LIN {X 0,Y 392.107,Z 460.199,A -85,B 0,C 180,E1 -19978.685,E2 -19978.685} C_VEL
LIN {X 0,Y 391.923,Z 458.619,A -85,B 0,C 180,E1 -19981.316,E2 -19981.316} C_VEL
LIN {X 0,Y 395.453,Z 464.321,A -85,B 0,C 180,E1 -19989.606,E2 -19989.606} C_VEL
LIN {X 0,Y 398.852,Z 469.35,A -85,B 0,C 180,E1 -19992.892,E2 -19992.892} C_VEL
LIN {X 0,Y 400.055,Z 470.705,A -85,B 0,C 180,E1 -19993.809,E2 -19993.809} C_VEL
LIN {X 0,Y 404.204,Z 476.438,A -85,B 0,C 180,E1 -19996.602,E2 -19996.602} C_VEL
LIN {X 0,Y 408.109,Z 481.813,A -85,B 0,C 180,E1 -19998.795,E2 -19998.795} C_VEL
LIN {X 0,Y 412.144,Z 487.49,A -85,B 0,C 180,E1 -20000.782,E2 -20000.782} C_VEL
LIN {X 0,Y 417.683,Z 495.416,A -85,B 0,C 180,E1 -20003.182,E2 -20003.182} C_VEL
LIN {X 0,Y 425.779,Z 507.797,A -85,B 0,C 180,E1 -20006.237,E2 -20006.237} C_VEL
LIN {X 0,Y 433.973,Z 521.148,A -85,B 0,C 180,E1 -20008.937,E2 -20008.937} C_VEL
LIN {X 0,Y 436.683,Z 526.126,A -85,B 0,C 180,E1 -20009.777,E2 -20009.777} C_VEL
LIN {X 0,Y 420.829,Z 746.012,A -85,B 0,C 180,E1 -20013.375,E2 -20013.375} C_VEL
LIN {X 0,Y 417.528,Z 772.58,A -85,B 0,C 180,E1 -20013.976,E2 -20013.976} C_VEL
LIN {X 0,Y 413.994,Z 793.305,A -85,B 0,C 180,E1 -20014.607,E2 -20014.607} C_VEL
LIN {X 0,Y 408.88,Z 817.43,A -85,B 0,C 180,E1 -20015.544,E2 -20015.544} C_VEL
LIN {X 0,Y 403.422,Z 838.547,A -85,B 0,C 180,E1 -20016.579,E2 -20016.579} C_VEL
LIN {X 0,Y 396.748,Z 861.148,A -85,B 0,C 180,E1 -20017.924,E2 -20017.924} C_VEL
LIN {X 0,Y 389.639,Z 881.774,A -85,B 0,C 180,E1 -20019.428,E2 -20019.428} C_VEL
LIN {X 0,Y 382.034,Z 901.996,A -85,B 0,C 180,E1 -20021.184,E2 -20021.184} C_VEL
LIN {X 0,Y 373.957,Z 921.227,A -85,B 0,C 180,E1 -20023.196,E2 -20023.196} C_VEL
LIN {X 0,Y 366.455,Z 937.947,A -85,B 0,C 180,E1 -20025.254,E2 -20025.254} C_VEL
LIN {X 0,Y 357.859,Z 955.928,A -85,B 0,C 180,E1 -20027.888,E2 -20027.888} C_VEL
LIN {X 0,Y 350.795,Z 969.964,A -85,B 0,C 180,E1 -20030.322,E2 -20030.322} C_VEL
LIN {X 0,Y 343.188,Z 984.792,A -85,B 0,C 180,E1 -20033.325,E2 -20033.325} C_VEL
LIN {X 0,Y 336.074,Z 998.178,A -85,B 0,C 180,E1 -20036.605,E2 -20036.605} C_VEL
LIN {X 0,Y 329.965,Z 1009.92,A -85,B 0,C 180,E1 -20040,E2 -20040} C_VEL
LIN {X 0,Y 324.125,Z 1021.359,A -85,B 0,C 180,E1 -20044.02,E2 -20044.02} C_VEL
LIN {X 0,Y 319.921,Z 1030.19,A -85,B 0,C 180,E1 -20047.779,E2 -20047.779} C_VEL
LIN {X 0,Y 316.256,Z 1038.778,A -85,B 0,C 180,E1 -20052.331,E2 -20052.331} C_VEL
LIN {X 0,Y 314.196,Z 1044.51,A -85,B 0,C 180,E1 -20056.192,E2 -20056.192} C_VEL
LIN {X 0,Y 312.799,Z 1049.554,A -85,B 0,C 180,E1 -20060.617,E2 -20060.617} C_VEL
LIN {X 0,Y 312.21,Z 1052.658,A -85,B 0,C 180,E1 -20064.671,E2 -20064.671} C_VEL
LIN {X 0,Y 312.029,Z 1054.407,A -85,B 0,C 180,E1 -20068.347,E2 -20068.347} C_VEL
LIN {X 0,Y 311.984,Z 1055.15,A -85,B 0,C 180,E1 -20072.204,E2 -20072.204} C_VEL
LIN {X 0,Y 312.068,Z 1054.525,A -85,B 0,C 180,E1 -20076.439,E2 -20076.439} C_VEL
LIN {X 0,Y 312.31,Z 1052.851,A -85,B 0,C 180,E1 -20080.142,E2 -20080.142} C_VEL
LIN {X 0,Y 312.996,Z 1049.964,A -85,B 0,C 180,E1 -20084.051,E2 -20084.051} C_VEL
LIN {X 0,Y 314.708,Z 1044.785,A -85,B 0,C 180,E1 -20088.771,E2 -20088.771} C_VEL
LIN {X 0,Y 317.043,Z 1039.138,A -85,B 0,C 180,E1 -20092.629,E2 -20092.629} C_VEL
LIN {X 0,Y 320.972,Z 1030.962,A -85,B 0,C 180,E1 -20097.053,E2 -20097.053} C_VEL
LIN {X 0,Y 325.565,Z 1022.129,A -85,B 0,C 180,E1 -20100.857,E2 -20100.857} C_VEL
LIN {X 0,Y 331.629,Z 1011.288,A -85,B 0,C 180,E1 -20104.74,E2 -20104.74} C_VEL
LIN {X 0,Y 338.541,Z 998.922,A -85,B 0,C 180,E1 -20108.334,E2 -20108.334} C_VEL
LIN {X 0,Y 346.21,Z 985.46,A -85,B 0,C 180,E1 -20111.626,E2 -20111.626} C_VEL
LIN {X 0,Y 354.624,Z 970.07,A -85,B 0,C 180,E1 -20114.721,E2 -20114.721} C_VEL
LIN {X 0,Y 363.408,Z 953.602,A -85,B 0,C 180,E1 -20117.509,E2 -20117.509} C_VEL
LIN {X 0,Y 372.16,Z 935.987,A -85,B 0,C 180,E1 -20119.971,E2 -20119.971} C_VEL
LIN {X 0,Y 380.693,Z 917.814,A -85,B 0,C 180,E1 -20122.117,E2 -20122.117} C_VEL
LIN {X 0,Y 389.097,Z 898.152,A -85,B 0,C 180,E1 -20124.045,E2 -20124.045} C_VEL
LIN {X 0,Y 396.341,Z 879.576,A -85,B 0,C 180,E1 -20125.584,E2 -20125.584} C_VEL
LIN {X 0,Y 404.502,Z 856.112,A -85,B 0,C 180,E1 -20127.187,E2 -20127.187} C_VEL
LIN {X 0,Y 408.136,Z 844.614,A -85,B 0,C 180,E1 -20127.862,E2 -20127.862} C_VEL
LIN {X 0,Y 409.545,Z 837.786,A -85,B 0,C 180,E1 -20128.344,E2 -20128.344} C_VEL
LIN {X 0,Y 411.055,Z 821.016,A -85,B 0,C 180,E1 -20129.882,E2 -20129.882} C_VEL
LIN {X 0,Y 412.236,Z 813.969,A -85,B 0,C 180,E1 -20130.298,E2 -20130.298} C_VEL
LIN {X 0,Y 417.189,Z 791.229,A -85,B 0,C 180,E1 -20131.12,E2 -20131.12} C_VEL
LIN {X 0,Y 421.292,Z 767.977,A -85,B 0,C 180,E1 -20131.778,E2 -20131.778} C_VEL
LIN {X 0,Y 424.228,Z 743.452,A -85,B 0,C 180,E1 -20132.284,E2 -20132.284} C_VEL
LIN {X 0,Y 440.243,Z 535.419,A -85,B 0,C 180,E1 -20135.639,E2 -20135.639} C_VEL
LIN {X 0,Y 432.705,Z 522.887,A -85,B 0,C 180,E1 -20138.372,E2 -20138.372} C_VEL
LIN {X 0,Y 425.772,Z 512.089,A -85,B 0,C 180,E1 -20141.268,E2 -20141.268} C_VEL
LIN {X 0,Y 420.737,Z 504.576,A -85,B 0,C 180,E1 -20143.714,E2 -20143.714} C_VEL
LIN {X 0,Y 417.623,Z 500.075,A -85,B 0,C 180,E1 -20145.44,E2 -20145.44} C_VEL
LIN {X 0,Y 414.64,Z 495.722,A -85,B 0,C 180,E1 -20147.324,E2 -20147.324} C_VEL
LIN {X 0,Y 411.54,Z 491.193,A -85,B 0,C 180,E1 -20149.642,E2 -20149.642} C_VEL
LIN {X 0,Y 408.5,Z 486.912,A -85,B 0,C 180,E1 -20152.546,E2 -20152.546} C_VEL
LIN {X 0,Y 407.925,Z 485.949,A -85,B 0,C 180,E1 -20153.243,E2 -20153.243} C_VEL
LIN {X 0,Y 404.96,Z 480.934,A -85,B 0,C 180,E1 -20160.707,E2 -20160.707} C_VEL
LIN {X 0,Y 405.174,Z 482.493,A -85,B 0,C 180,E1 -20163.395,E2 -20163.395} C_VEL
LIN {X 0,Y 408.31,Z 486.414,A -85,B 0,C 180,E1 -20168.875,E2 -20168.875} C_VEL
LIN {X 0,Y 410.739,Z 490.415,A -85,B 0,C 180,E1 -20171.372,E2 -20171.372} C_VEL
LIN {X 0,Y 412.175,Z 492.139,A -85,B 0,C 180,E1 -20172.54,E2 -20172.54} C_VEL
LIN {X 0,Y 416.043,Z 497.712,A -85,B 0,C 180,E1 -20175.258,E2 -20175.258} C_VEL
LIN {X 0,Y 419.58,Z 502.842,A -85,B 0,C 180,E1 -20177.331,E2 -20177.331} C_VEL
LIN {X 0,Y 423.084,Z 508.142,A -85,B 0,C 180,E1 -20179.142,E2 -20179.142} C_VEL
LIN {X 0,Y 430.274,Z 520.703,A -85,B 0,C 180,E1 -20182.403,E2 -20182.403} C_VEL
LIN {X 0,Y 438.135,Z 535.607,A -85,B 0,C 180,E1 -20185.443,E2 -20185.443} C_VEL
LIN {X 0,Y 440.062,Z 539.907,A -85,B 0,C 180,E1 -20186.145,E2 -20186.145} C_VEL
LIN {X 0,Y 423.319,Z 757.439,A -85,B 0,C 180,E1 -20189.661,E2 -20189.661} C_VEL
LIN {X 0,Y 419.717,Z 784.19,A -85,B 0,C 180,E1 -20190.228,E2 -20190.228} C_VEL
LIN {X 0,Y 415.608,Z 805.997,A -85,B 0,C 180,E1 -20190.833,E2 -20190.833} C_VEL
LIN {X 0,Y 409.689,Z 831.066,A -85,B 0,C 180,E1 -20191.743,E2 -20191.743} C_VEL
LIN {X 0,Y 403.918,Z 851.482,A -85,B 0,C 180,E1 -20192.684,E2 -20192.684} C_VEL
LIN {X 0,Y 396.612,Z 874.086,A -85,B 0,C 180,E1 -20193.959,E2 -20193.959} C_VEL
LIN {X 0,Y 389.187,Z 894.048,A -85,B 0,C 180,E1 -20195.342,E2 -20195.342} C_VEL
LIN {X 0,Y 381.105,Z 913.869,A -85,B 0,C 180,E1 -20196.974,E2 -20196.974} C_VEL
LIN {X 0,Y 372.228,Z 933.564,A -85,B 0,C 180,E1 -20198.946,E2 -20198.946} C_VEL
LIN {X 0,Y 364.051,Z 950.448,A -85,B 0,C 180,E1 -20200.948,E2 -20200.948} C_VEL
LIN {X 0,Y 354.07,Z 969.767,A -85,B 0,C 180,E1 -20203.702,E2 -20203.702} C_VEL
LIN {X 0,Y 345.849,Z 984.889,A -85,B 0,C 180,E1 -20206.292,E2 -20206.292} C_VEL
LIN {X 0,Y 336.675,Z 1001.243,A -85,B 0,C 180,E1 -20209.651,E2 -20209.651} C_VEL
LIN {X 0,Y 329.367,Z 1014.076,A -85,B 0,C 180,E1 -20212.834,E2 -20212.834} C_VEL
LIN {X 0,Y 322.102,Z 1027.018,A -85,B 0,C 180,E1 -20216.67,E2 -20216.67} C_VEL
LIN {X 0,Y 316.389,Z 1037.489,A -85,B 0,C 180,E1 -20220.461,E2 -20220.461} C_VEL
LIN {X 0,Y 311.489,Z 1047.292,A -85,B 0,C 180,E1 -20224.727,E2 -20224.727} C_VEL
LIN {X 0,Y 307.959,Z 1055.162,A -85,B 0,C 180,E1 -20229.075,E2 -20229.075} C_VEL
LIN {X 0,Y 305.682,Z 1061.542,A -85,B 0,C 180,E1 -20233.466,E2 -20233.466} C_VEL
LIN {X 0,Y 304.419,Z 1066.404,A -85,B 0,C 180,E1 -20238.058,E2 -20238.058} C_VEL
LIN {X 0,Y 304.013,Z 1069.246,A -85,B 0,C 180,E1 -20241.885,E2 -20241.885} C_VEL
LIN {X 0,Y 303.96,Z 1071.045,A -85,B 0,C 180,E1 -20245.85,E2 -20245.85} C_VEL
LIN {X 0,Y 304.002,Z 1071.567,A -85,B 0,C 180,E1 -20250,E2 -20250} C_VEL
LIN {X 0,Y 303.97,Z 1070.824,A -85,B 0,C 180,E1 -20253.772,E2 -20253.772} C_VEL
LIN {X 0,Y 304.002,Z 1069.099,A -85,B 0,C 180,E1 -20257.37,E2 -20257.37} C_VEL
LIN {X 0,Y 304.317,Z 1066.031,A -85,B 0,C 180,E1 -20261.37,E2 -20261.37} C_VEL
LIN {X 0,Y 305.49,Z 1060.637,A -85,B 0,C 180,E1 -20266.153,E2 -20266.153} C_VEL
LIN {X 0,Y 307.385,Z 1054.653,A -85,B 0,C 180,E1 -20270.17,E2 -20270.17} C_VEL
LIN {X 0,Y 310.78,Z 1046.13,A -85,B 0,C 180,E1 -20274.724,E2 -20274.724} C_VEL
LIN {X 0,Y 314.948,Z 1036.991,A -85,B 0,C 180,E1 -20278.646,E2 -20278.646} C_VEL
LIN {X 0,Y 320.569,Z 1025.802,A -85,B 0,C 180,E1 -20282.657,E2 -20282.657} C_VEL
LIN {X 0,Y 327.144,Z 1013.096,A -85,B 0,C 180,E1 -20286.366,E2 -20286.366} C_VEL
LIN {X 0,Y 334.671,Z 998.993,A -85,B 0,C 180,E1 -20289.84,E2 -20289.84} C_VEL
LIN {X 0,Y 342.892,Z 983.203,A -85,B 0,C 180,E1 -20293.028,E2 -20293.028} C_VEL
LIN {X 0,Y 351.564,Z 966.327,A -85,B 0,C 180,E1 -20295.901,E2 -20295.901} C_VEL
LIN {X 0,Y 359.956,Z 948.899,A -85,B 0,C 180,E1 -20298.351,E2 -20298.351} C_VEL
LIN {X 0,Y 367.87,Z 931.67,A -85,B 0,C 180,E1 -20300.41,E2 -20300.41} C_VEL
LIN {X 0,Y 376.774,Z 910.555,A -85,B 0,C 180,E1 -20302.513,E2 -20302.513} C_VEL
LIN {X 0,Y 383.859,Z 892.297,A -85,B 0,C 180,E1 -20304.028,E2 -20304.028} C_VEL
LIN {X 0,Y 391.912,Z 869.15,A -85,B 0,C 180,E1 -20305.624,E2 -20305.624} C_VEL
LIN {X 0,Y 397.756,Z 850.018,A -85,B 0,C 180,E1 -20306.704,E2 -20306.704} C_VEL
LIN {X 0,Y 403.893,Z 827.253,A -85,B 0,C 180,E1 -20307.764,E2 -20307.764} C_VEL
LIN {X 0,Y 409.005,Z 803.859,A -85,B 0,C 180,E1 -20308.606,E2 -20308.606} C_VEL
LIN {X 0,Y 413.132,Z 780.688,A -85,B 0,C 180,E1 -20309.254,E2 -20309.254} C_VEL
LIN {X 0,Y 416.173,Z 755.582,A -85,B 0,C 180,E1 -20309.781,E2 -20309.781} C_VEL
LIN {X 0,Y 432.44,Z 534.422,A -85,B 0,C 180,E1 -20313.402,E2 -20313.402} C_VEL
LIN {X 0,Y 425.765,Z 521.335,A -85,B 0,C 180,E1 -20315.66,E2 -20315.66} C_VEL
LIN {X 0,Y 419.365,Z 509.666,A -85,B 0,C 180,E1 -20318.054,E2 -20318.054} C_VEL
LIN {X 0,Y 413.828,Z 500.099,A -85,B 0,C 180,E1 -20320.376,E2 -20320.376} C_VEL
LIN {X 0,Y 408.544,Z 492.288,A -85,B 0,C 180,E1 -20322.847,E2 -20322.847} C_VEL
LIN {X 0,Y 404.593,Z 486.761,A -85,B 0,C 180,E1 -20324.96,E2 -20324.96} C_VEL
LIN {X 0,Y 401.658,Z 482.574,A -85,B 0,C 180,E1 -20326.76,E2 -20326.76} C_VEL
LIN {X 0,Y 397.969,Z 477.456,A -85,B 0,C 180,E1 -20329.431,E2 -20329.431} C_VEL
LIN {X 0,Y 395.072,Z 473.702,A -85,B 0,C 180,E1 -20332.072,E2 -20332.072} C_VEL
LIN {X 0,Y 394.278,Z 472.195,A -85,B 0,C 180,E1 -20333.008,E2 -20333.008} C_VEL
LIN {X 0,Y 390.943,Z 466.591,A -85,B 0,C 180,E1 -20341.172,E2 -20341.172} C_VEL
LIN {X 0,Y 391.332,Z 468.804,A -85,B 0,C 180,E1 -20344.543,E2 -20344.543} C_VEL
LIN {X 0,Y 394.595,Z 472.62,A -85,B 0,C 180,E1 -20349.775,E2 -20349.775} C_VEL
LIN {X 0,Y 397.351,Z 476.896,A -85,B 0,C 180,E1 -20352.498,E2 -20352.498} C_VEL
LIN {X 0,Y 398.703,Z 478.42,A -85,B 0,C 180,E1 -20353.561,E2 -20353.561} C_VEL
LIN {X 0,Y 402.767,Z 484.173,A -85,B 0,C 180,E1 -20356.366,E2 -20356.366} C_VEL
LIN {X 0,Y 406.481,Z 489.377,A -85,B 0,C 180,E1 -20358.501,E2 -20358.501} C_VEL
LIN {X 0,Y 410.443,Z 495.07,A -85,B 0,C 180,E1 -20360.499,E2 -20360.499} C_VEL
LIN {X 0,Y 415.829,Z 502.974,A -85,B 0,C 180,E1 -20362.889,E2 -20362.889} C_VEL
LIN {X 0,Y 423.519,Z 514.987,A -85,B 0,C 180,E1 -20365.86,E2 -20365.86} C_VEL
LIN {X 0,Y 431.288,Z 527.889,A -85,B 0,C 180,E1 -20368.49,E2 -20368.49} C_VEL
LIN {X 0,Y 432.587,Z 530.46,A -85,B 0,C 180,E1 -20368.913,E2 -20368.913} C_VEL
LIN {X 0,Y 416.611,Z 746.198,A -85,B 0,C 180,E1 -20372.444,E2 -20372.444} C_VEL
LIN {X 0,Y 413.237,Z 772.776,A -85,B 0,C 180,E1 -20373.044,E2 -20373.044} C_VEL
LIN {X 0,Y 409.644,Z 793.399,A -85,B 0,C 180,E1 -20373.668,E2 -20373.668} C_VEL
LIN {X 0,Y 404.466,Z 817.349,A -85,B 0,C 180,E1 -20374.592,E2 -20374.592} C_VEL
LIN {X 0,Y 399.02,Z 837.987,A -85,B 0,C 180,E1 -20375.595,E2 -20375.595} C_VEL
LIN {X 0,Y 392.484,Z 859.751,A -85,B 0,C 180,E1 -20376.875,E2 -20376.875} C_VEL
LIN {X 0,Y 385.178,Z 880.634,A -85,B 0,C 180,E1 -20378.375,E2 -20378.375} C_VEL
LIN {X 0,Y 378.164,Z 898.884,A -85,B 0,C 180,E1 -20379.935,E2 -20379.935} C_VEL
LIN {X 0,Y 369.204,Z 920.008,A -85,B 0,C 180,E1 -20382.093,E2 -20382.093} C_VEL
LIN {X 0,Y 361.513,Z 936.692,A -85,B 0,C 180,E1 -20384.132,E2 -20384.132} C_VEL
LIN {X 0,Y 352.516,Z 955.067,A -85,B 0,C 180,E1 -20386.8,E2 -20386.8} C_VEL
LIN {X 0,Y 344.576,Z 970.313,A -85,B 0,C 180,E1 -20389.458,E2 -20389.458} C_VEL
LIN {X 0,Y 336.694,Z 985.124,A -85,B 0,C 180,E1 -20392.498,E2 -20392.498} C_VEL
LIN {X 0,Y 328.953,Z 999.119,A -85,B 0,C 180,E1 -20395.993,E2 -20395.993} C_VEL
LIN {X 0,Y 322.348,Z 1011.352,A -85,B 0,C 180,E1 -20399.628,E2 -20399.628} C_VEL
LIN {X 0,Y 316.58,Z 1022.099,A -85,B 0,C 180,E1 -20403.555,E2 -20403.555} C_VEL
LIN {X 0,Y 312.039,Z 1031.265,A -85,B 0,C 180,E1 -20407.585,E2 -20407.585} C_VEL
LIN {X 0,Y 308.405,Z 1039.339,A -85,B 0,C 180,E1 -20412.061,E2 -20412.061} C_VEL
LIN {X 0,Y 306.264,Z 1045.015,A -85,B 0,C 180,E1 -20416.019,E2 -20416.019} C_VEL
LIN {X 0,Y 304.773,Z 1050.105,A -85,B 0,C 180,E1 -20420.749,E2 -20420.749} C_VEL
LIN {X 0,Y 304.21,Z 1053,A -85,B 0,C 180,E1 -20424.72,E2 -20424.72} C_VEL
LIN {X 0,Y 304.03,Z 1054.698,A -85,B 0,C 180,E1 -20428.492,E2 -20428.492} C_VEL
LIN {X 0,Y 303.99,Z 1055.394,A -85,B 0,C 180,E1 -20432.639,E2 -20432.639} C_VEL
LIN {X 0,Y 304.084,Z 1054.663,A -85,B 0,C 180,E1 -20436.798,E2 -20436.798} C_VEL
LIN {X 0,Y 304.342,Z 1053.049,A -85,B 0,C 180,E1 -20440.41,E2 -20440.41} C_VEL
LIN {X 0,Y 305.096,Z 1050.156,A -85,B 0,C 180,E1 -20444.423,E2 -20444.423} C_VEL
LIN {X 0,Y 306.918,Z 1045.034,A -85,B 0,C 180,E1 -20449.211,E2 -20449.211} C_VEL
LIN {X 0,Y 309.449,Z 1039.309,A -85,B 0,C 180,E1 -20453.216,E2 -20453.216} C_VEL
LIN {X 0,Y 313.625,Z 1031.117,A -85,B 0,C 180,E1 -20457.741,E2 -20457.741} C_VEL
LIN {X 0,Y 318.474,Z 1022.276,A -85,B 0,C 180,E1 -20461.622,E2 -20461.622} C_VEL
LIN {X 0,Y 324.84,Z 1011.42,A -85,B 0,C 180,E1 -20465.574,E2 -20465.574} C_VEL
LIN {X 0,Y 332.074,Z 999.042,A -85,B 0,C 180,E1 -20469.222,E2 -20469.222} C_VEL
LIN {X 0,Y 340.062,Z 985.569,A -85,B 0,C 180,E1 -20472.553,E2 -20472.553} C_VEL
LIN {X 0,Y 348.532,Z 970.629,A -85,B 0,C 180,E1 -20475.59,E2 -20475.59} C_VEL
LIN {X 0,Y 356.861,Z 955.523,A -85,B 0,C 180,E1 -20478.185,E2 -20478.185} C_VEL
LIN {X 0,Y 366.378,Z 937.141,A -85,B 0,C 180,E1 -20480.811,E2 -20480.811} C_VEL
LIN {X 0,Y 374.547,Z 920.273,A -85,B 0,C 180,E1 -20482.833,E2 -20482.833} C_VEL
LIN {X 0,Y 384.052,Z 898.875,A -85,B 0,C 180,E1 -20484.966,E2 -20484.966} C_VEL
LIN {X 0,Y 391.16,Z 881.166,A -85,B 0,C 180,E1 -20486.442,E2 -20486.442} C_VEL
LIN {X 0,Y 399.138,Z 859.19,A -85,B 0,C 180,E1 -20487.973,E2 -20487.973} C_VEL
LIN {X 0,Y 405.748,Z 837.99,A -85,B 0,C 180,E1 -20489.183,E2 -20489.183} C_VEL
LIN {X 0,Y 411.995,Z 815.05,A -85,B 0,C 180,E1 -20490.255,E2 -20490.255} C_VEL
LIN {X 0,Y 412.236,Z 813.969,A -85,B 0,C 180,E1 -20490.298,E2 -20490.298} C_VEL
LIN {X 0,Y 413.356,Z 806.832,A -85,B 0,C 180,E1 -20490.698,E2 -20490.698} C_VEL
LIN {X 0,Y 414.24,Z 789.235,A -85,B 0,C 180,E1 -20492.044,E2 -20492.044} C_VEL
LIN {X 0,Y 415.089,Z 781.926,A -85,B 0,C 180,E1 -20492.378,E2 -20492.378} C_VEL
LIN {X 0,Y 418.675,Z 758.825,A -85,B 0,C 180,E1 -20492.947,E2 -20492.947} C_VEL
LIN {X 0,Y 421.397,Z 733.209,A -85,B 0,C 180,E1 -20493.422,E2 -20493.422} C_VEL
LIN {X 0,Y 436.472,Z 540.091,A -85,B 0,C 180,E1 -20496.527,E2 -20496.527} C_VEL
LIN {X 0,Y 430.16,Z 529.414,A -85,B 0,C 180,E1 -20498.917,E2 -20498.917} C_VEL
LIN {X 0,Y 423.64,Z 519,A -85,B 0,C 180,E1 -20501.74,E2 -20501.74} C_VEL
LIN {X 0,Y 418.868,Z 511.764,A -85,B 0,C 180,E1 -20504.138,E2 -20504.138} C_VEL
LIN {X 0,Y 415.843,Z 507.313,A -85,B 0,C 180,E1 -20505.874,E2 -20505.874} C_VEL
LIN {X 0,Y 413.255,Z 503.408,A -85,B 0,C 180,E1 -20507.564,E2 -20507.564} C_VEL
LIN {X 0,Y 410.054,Z 498.749,A -85,B 0,C 180,E1 -20510.03,E2 -20510.03} C_VEL
LIN {X 0,Y 407.172,Z 494.337,A -85,B 0,C 180,E1 -20512.947,E2 -20512.947} C_VEL
LIN {X 0,Y 403.983,Z 488.887,A -85,B 0,C 180,E1 -20520.709,E2 -20520.709} C_VEL
LIN {X 0,Y 404.263,Z 490.703,A -85,B 0,C 180,E1 -20523.687,E2 -20523.687} C_VEL
LIN {X 0,Y 407.205,Z 494.378,A -85,B 0,C 180,E1 -20528.757,E2 -20528.757} C_VEL
LIN {X 0,Y 409.769,Z 498.475,A -85,B 0,C 180,E1 -20531.4,E2 -20531.4} C_VEL
LIN {X 0,Y 410.93,Z 499.999,A -85,B 0,C 180,E1 -20532.364,E2 -20532.364} C_VEL
LIN {X 0,Y 414.531,Z 505.26,A -85,B 0,C 180,E1 -20534.957,E2 -20534.957} C_VEL
LIN {X 0,Y 417.988,Z 510.399,A -85,B 0,C 180,E1 -20537.04,E2 -20537.04} C_VEL
LIN {X 0,Y 421.29,Z 515.524,A -85,B 0,C 180,E1 -20538.795,E2 -20538.795} C_VEL
LIN {X 0,Y 428.233,Z 527.953,A -85,B 0,C 180,E1 -20542.034,E2 -20542.034} C_VEL
LIN {X 0,Y 435.709,Z 542.535,A -85,B 0,C 180,E1 -20545.013,E2 -20545.013} C_VEL
LIN {X 0,Y 436.342,Z 544.175,A -85,B 0,C 180,E1 -20545.261,E2 -20545.261} C_VEL
LIN {X 0,Y 419.514,Z 757.283,A -85,B 0,C 180,E1 -20548.7,E2 -20548.7} C_VEL
LIN {X 0,Y 415.84,Z 784.009,A -85,B 0,C 180,E1 -20549.263,E2 -20549.263} C_VEL
LIN {X 0,Y 411.668,Z 805.744,A -85,B 0,C 180,E1 -20549.862,E2 -20549.862} C_VEL
LIN {X 0,Y 405.695,Z 830.577,A -85,B 0,C 180,E1 -20550.753,E2 -20550.753} C_VEL
LIN {X 0,Y 399.826,Z 850.919,A -85,B 0,C 180,E1 -20551.68,E2 -20551.68} C_VEL
LIN {X 0,Y 392.489,Z 873.21,A -85,B 0,C 180,E1 -20552.921,E2 -20552.921} C_VEL
LIN {X 0,Y 384.643,Z 893.826,A -85,B 0,C 180,E1 -20554.34,E2 -20554.34} C_VEL
LIN {X 0,Y 376.465,Z 913.378,A -85,B 0,C 180,E1 -20555.943,E2 -20555.943} C_VEL
LIN {X 0,Y 367.131,Z 933.544,A -85,B 0,C 180,E1 -20557.958,E2 -20557.958} C_VEL
LIN {X 0,Y 358.732,Z 950.377,A -85,B 0,C 180,E1 -20559.959,E2 -20559.959} C_VEL
LIN {X 0,Y 348.439,Z 969.671,A -85,B 0,C 180,E1 -20562.725,E2 -20562.725} C_VEL
LIN {X 0,Y 340.417,Z 983.933,A -85,B 0,C 180,E1 -20565.175,E2 -20565.175} C_VEL
LIN {X 0,Y 331.284,Z 999.705,A -85,B 0,C 180,E1 -20568.394,E2 -20568.394} C_VEL
LIN {X 0,Y 323.557,Z 1012.659,A -85,B 0,C 180,E1 -20571.6,E2 -20571.6} C_VEL
LIN {X 0,Y 316.145,Z 1025.308,A -85,B 0,C 180,E1 -20575.318,E2 -20575.318} C_VEL
LIN {X 0,Y 309.724,Z 1036.399,A -85,B 0,C 180,E1 -20579.331,E2 -20579.331} C_VEL
LIN {X 0,Y 304.832,Z 1045.506,A -85,B 0,C 180,E1 -20583.296,E2 -20583.296} C_VEL
LIN {X 0,Y 300.554,Z 1054.364,A -85,B 0,C 180,E1 -20588.124,E2 -20588.124} C_VEL
LIN {X 0,Y 298.169,Z 1060.337,A -85,B 0,C 180,E1 -20592.247,E2 -20592.247} C_VEL
LIN {X 0,Y 296.588,Z 1065.714,A -85,B 0,C 180,E1 -20597.144,E2 -20597.144} C_VEL
LIN {X 0,Y 296.057,Z 1068.802,A -85,B 0,C 180,E1 -20601.258,E2 -20601.258} C_VEL
LIN {X 0,Y 295.965,Z 1070.558,A -85,B 0,C 180,E1 -20604.961,E2 -20604.961} C_VEL
LIN {X 0,Y 295.988,Z 1071.34,A -85,B 0,C 180,E1 -20608.839,E2 -20608.839} C_VEL
LIN {X 0,Y 295.982,Z 1070.949,A -85,B 0,C 180,E1 -20612.905,E2 -20612.905} C_VEL
LIN {X 0,Y 295.985,Z 1069.219,A -85,B 0,C 180,E1 -20616.985,E2 -20616.985} C_VEL
LIN {X 0,Y 296.236,Z 1066.514,A -85,B 0,C 180,E1 -20620.82,E2 -20620.82} C_VEL
LIN {X 0,Y 297.163,Z 1062.133,A -85,B 0,C 180,E1 -20625.216,E2 -20625.216} C_VEL
LIN {X 0,Y 299.206,Z 1055.636,A -85,B 0,C 180,E1 -20629.93,E2 -20629.93} C_VEL
LIN {X 0,Y 302.078,Z 1048.532,A -85,B 0,C 180,E1 -20634.025,E2 -20634.025} C_VEL
LIN {X 0,Y 306.759,Z 1038.581,A -85,B 0,C 180,E1 -20638.63,E2 -20638.63} C_VEL
LIN {X 0,Y 311.855,Z 1028.689,A -85,B 0,C 180,E1 -20642.374,E2 -20642.374} C_VEL
LIN {X 0,Y 319.086,Z 1015.375,A -85,B 0,C 180,E1 -20646.54,E2 -20646.54} C_VEL
LIN {X 0,Y 326.141,Z 1002.551,A -85,B 0,C 180,E1 -20649.848,E2 -20649.848} C_VEL
LIN {X 0,Y 334.628,Z 987.115,A -85,B 0,C 180,E1 -20653.19,E2 -20653.19} C_VEL
LIN {X 0,Y 342.594,Z 972.097,A -85,B 0,C 180,E1 -20655.887,E2 -20655.887} C_VEL
LIN {X 0,Y 351.575,Z 954.674,A -85,B 0,C 180,E1 -20658.539,E2 -20658.539} C_VEL
LIN {X 0,Y 360.377,Z 936.242,A -85,B 0,C 180,E1 -20660.85,E2 -20660.85} C_VEL
LIN {X 0,Y 368.441,Z 918.26,A -85,B 0,C 180,E1 -20662.758,E2 -20662.758} C_VEL
LIN {X 0,Y 377.103,Z 897.095,A -85,B 0,C 180,E1 -20664.621,E2 -20664.621} C_VEL
LIN {X 0,Y 384.111,Z 878.167,A -85,B 0,C 180,E1 -20666.006,E2 -20666.006} C_VEL
LIN {X 0,Y 391.773,Z 854.86,A -85,B 0,C 180,E1 -20667.417,E2 -20667.417} C_VEL
LIN {X 0,Y 397.76,Z 833.621,A -85,B 0,C 180,E1 -20668.449,E2 -20668.449} C_VEL
LIN {X 0,Y 403.532,Z 809.714,A -85,B 0,C 180,E1 -20669.379,E2 -20669.379} C_VEL
LIN {X 0,Y 407.972,Z 786.31,A -85,B 0,C 180,E1 -20670.064,E2 -20670.064} C_VEL
LIN {X 0,Y 411.49,Z 761.683,A -85,B 0,C 180,E1 -20670.621,E2 -20670.621} C_VEL
LIN {X 0,Y 415.66,Z 708.814,A -85,B 0,C 180,E1 -20671.518,E2 -20671.518} C_VEL
LIN {X 0,Y 428.389,Z 538.48,A -85,B 0,C 180,E1 -20674.303,E2 -20674.303} C_VEL
LIN {X 0,Y 422.76,Z 527.263,A -85,B 0,C 180,E1 -20676.292,E2 -20676.292} C_VEL
LIN {X 0,Y 416.946,Z 516.392,A -85,B 0,C 180,E1 -20678.548,E2 -20678.548} C_VEL
LIN {X 0,Y 411.771,Z 507.237,A -85,B 0,C 180,E1 -20680.79,E2 -20680.79} C_VEL
LIN {X 0,Y 406.611,Z 499.485,A -85,B 0,C 180,E1 -20683.279,E2 -20683.279} C_VEL
LIN {X 0,Y 402.77,Z 493.992,A -85,B 0,C 180,E1 -20685.405,E2 -20685.405} C_VEL
LIN {X 0,Y 400.136,Z 490.146,A -85,B 0,C 180,E1 -20687.076,E2 -20687.076} C_VEL
LIN {X 0,Y 396.634,Z 485.178,A -85,B 0,C 180,E1 -20689.689,E2 -20689.689} C_VEL
LIN {X 0,Y 393.764,Z 481.254,A -85,B 0,C 180,E1 -20692.412,E2 -20692.412} C_VEL
LIN {X 0,Y 393.175,Z 480.083,A -85,B 0,C 180,E1 -20693.135,E2 -20693.135} C_VEL
LIN {X 0,Y 389.968,Z 474.534,A -85,B 0,C 180,E1 -20701.175,E2 -20701.175} C_VEL
LIN {X 0,Y 390.545,Z 477.299,A -85,B 0,C 180,E1 -20705.141,E2 -20705.141} C_VEL
LIN {X 0,Y 393.421,Z 480.441,A -85,B 0,C 180,E1 -20709.575,E2 -20709.575} C_VEL
LIN {X 0,Y 396.332,Z 484.908,A -85,B 0,C 180,E1 -20712.487,E2 -20712.487} C_VEL
LIN {X 0,Y 397.53,Z 486.454,A -85,B 0,C 180,E1 -20713.454,E2 -20713.454} C_VEL
LIN {X 0,Y 401.23,Z 491.726,A -85,B 0,C 180,E1 -20716.059,E2 -20716.059} C_VEL
LIN {X 0,Y 404.987,Z 497.134,A -85,B 0,C 180,E1 -20718.274,E2 -20718.274} C_VEL
LIN {X 0,Y 408.822,Z 502.749,A -85,B 0,C 180,E1 -20720.248,E2 -20720.248} C_VEL
LIN {X 0,Y 414.357,Z 511.11,A -85,B 0,C 180,E1 -20722.75,E2 -20722.75} C_VEL
LIN {X 0,Y 421.363,Z 522.322,A -85,B 0,C 180,E1 -20725.512,E2 -20725.512} C_VEL
LIN {X 0,Y 428.604,Z 534.588,A -85,B 0,C 180,E1 -20728.03,E2 -20728.03} C_VEL
LIN {X 0,Y 412.497,Z 746.49,A -85,B 0,C 180,E1 -20731.496,E2 -20731.496} C_VEL
LIN {X 0,Y 409.037,Z 773.102,A -85,B 0,C 180,E1 -20732.095,E2 -20732.095} C_VEL
LIN {X 0,Y 405.349,Z 793.792,A -85,B 0,C 180,E1 -20732.72,E2 -20732.72} C_VEL
LIN {X 0,Y 399.987,Z 817.951,A -85,B 0,C 180,E1 -20733.65,E2 -20733.65} C_VEL
LIN {X 0,Y 394.419,Z 838.544,A -85,B 0,C 180,E1 -20734.65,E2 -20734.65} C_VEL
LIN {X 0,Y 387.513,Z 860.948,A -85,B 0,C 180,E1 -20735.971,E2 -20735.971} C_VEL
LIN {X 0,Y 379.937,Z 881.899,A -85,B 0,C 180,E1 -20737.49,E2 -20737.49} C_VEL
LIN {X 0,Y 372.171,Z 901.502,A -85,B 0,C 180,E1 -20739.186,E2 -20739.186} C_VEL
LIN {X 0,Y 363.281,Z 921.613,A -85,B 0,C 180,E1 -20741.288,E2 -20741.288} C_VEL
LIN {X 0,Y 355.136,Z 938.722,A -85,B 0,C 180,E1 -20743.414,E2 -20743.414} C_VEL
LIN {X 0,Y 345.986,Z 956.649,A -85,B 0,C 180,E1 -20746.085,E2 -20746.085} C_VEL
LIN {X 0,Y 337.988,Z 971.495,A -85,B 0,C 180,E1 -20748.722,E2 -20748.722} C_VEL
LIN {X 0,Y 329.044,Z 987.524,A -85,B 0,C 180,E1 -20752.133,E2 -20752.133} C_VEL
LIN {X 0,Y 321.873,Z 1000.061,A -85,B 0,C 180,E1 -20755.355,E2 -20755.355} C_VEL
LIN {X 0,Y 314.734,Z 1012.678,A -85,B 0,C 180,E1 -20759.237,E2 -20759.237} C_VEL
LIN {X 0,Y 309.057,Z 1022.838,A -85,B 0,C 180,E1 -20763.068,E2 -20763.068} C_VEL
LIN {X 0,Y 304.159,Z 1032.324,A -85,B 0,C 180,E1 -20767.38,E2 -20767.38} C_VEL
LIN {X 0,Y 300.562,Z 1039.899,A -85,B 0,C 180,E1 -20771.777,E2 -20771.777} C_VEL
LIN {X 0,Y 298.255,Z 1045.767,A -85,B 0,C 180,E1 -20776.032,E2 -20776.032} C_VEL
LIN {X 0,Y 296.76,Z 1050.611,A -85,B 0,C 180,E1 -20780.832,E2 -20780.832} C_VEL
LIN {X 0,Y 296.211,Z 1053.343,A -85,B 0,C 180,E1 -20784.771,E2 -20784.771} C_VEL
LIN {X 0,Y 296.025,Z 1055.073,A -85,B 0,C 180,E1 -20788.889,E2 -20788.889} C_VEL
LIN {X 0,Y 295.998,Z 1055.538,A -85,B 0,C 180,E1 -20793.292,E2 -20793.292} C_VEL
LIN {X 0,Y 296.102,Z 1054.801,A -85,B 0,C 180,E1 -20797.178,E2 -20797.178} C_VEL
LIN {X 0,Y 296.423,Z 1053.071,A -85,B 0,C 180,E1 -20801.007,E2 -20801.007} C_VEL
LIN {X 0,Y 297.44,Z 1049.704,A -85,B 0,C 180,E1 -20805.601,E2 -20805.601} C_VEL
LIN {X 0,Y 299.388,Z 1044.714,A -85,B 0,C 180,E1 -20810.121,E2 -20810.121} C_VEL
LIN {X 0,Y 302.353,Z 1038.587,A -85,B 0,C 180,E1 -20814.417,E2 -20814.417} C_VEL
LIN {X 0,Y 306.965,Z 1030.074,A -85,B 0,C 180,E1 -20819.035,E2 -20819.035} C_VEL
LIN {X 0,Y 312.001,Z 1021.516,A -85,B 0,C 180,E1 -20822.793,E2 -20822.793} C_VEL
LIN {X 0,Y 319.464,Z 1009.275,A -85,B 0,C 180,E1 -20827.162,E2 -20827.162} C_VEL
LIN {X 0,Y 326.479,Z 997.901,A -85,B 0,C 180,E1 -20830.487,E2 -20830.487} C_VEL
LIN {X 0,Y 335.765,Z 982.636,A -85,B 0,C 180,E1 -20834.174,E2 -20834.174} C_VEL
LIN {X 0,Y 343.775,Z 969.032,A -85,B 0,C 180,E1 -20836.89,E2 -20836.89} C_VEL
LIN {X 0,Y 353.545,Z 951.748,A -85,B 0,C 180,E1 -20839.783,E2 -20839.783} C_VEL
LIN {X 0,Y 362.382,Z 934.969,A -85,B 0,C 180,E1 -20842.105,E2 -20842.105} C_VEL
LIN {X 0,Y 371.769,Z 915.98,A -85,B 0,C 180,E1 -20844.316,E2 -20844.316} C_VEL
LIN {X 0,Y 380.361,Z 896.66,A -85,B 0,C 180,E1 -20846.171,E2 -20846.171} C_VEL
LIN {X 0,Y 388.68,Z 876.258,A -85,B 0,C 180,E1 -20847.818,E2 -20847.818} C_VEL
LIN {X 0,Y 396.269,Z 854.919,A -85,B 0,C 180,E1 -20849.224,E2 -20849.224} C_VEL
LIN {X 0,Y 402.897,Z 833.756,A -85,B 0,C 180,E1 -20850.387,E2 -20850.387} C_VEL
LIN {X 0,Y 409.117,Z 810.129,A -85,B 0,C 180,E1 -20851.426,E2 -20851.426} C_VEL
LIN {X 0,Y 413.805,Z 788.624,A -85,B 0,C 180,E1 -20852.175,E2 -20852.175} C_VEL
LIN {X 0,Y 415.089,Z 781.926,A -85,B 0,C 180,E1 -20852.378,E2 -20852.378} C_VEL
LIN {X 0,Y 415.873,Z 774.545,A -85,B 0,C 180,E1 -20852.694,E2 -20852.694} C_VEL
LIN {X 0,Y 415.898,Z 755.236,A -85,B 0,C 180,E1 -20853.908,E2 -20853.908} C_VEL
LIN {X 0,Y 416.266,Z 748.791,A -85,B 0,C 180,E1 -20854.126,E2 -20854.126} C_VEL
LIN {X 0,Y 422.531,Z 672.842,A -85,B 0,C 180,E1 -20855.369,E2 -20855.369} C_VEL
LIN {X 0,Y 432.857,Z 544.806,A -85,B 0,C 180,E1 -20857.413,E2 -20857.413} C_VEL
LIN {X 0,Y 425.931,Z 532.993,A -85,B 0,C 180,E1 -20860.206,E2 -20860.206} C_VEL
LIN {X 0,Y 420.009,Z 523.559,A -85,B 0,C 180,E1 -20862.973,E2 -20862.973} C_VEL
LIN {X 0,Y 415.196,Z 516.036,A -85,B 0,C 180,E1 -20865.638,E2 -20865.638} C_VEL
LIN {X 0,Y 411.681,Z 510.855,A -85,B 0,C 180,E1 -20867.943,E2 -20867.943} C_VEL
LIN {X 0,Y 408.914,Z 506.631,A -85,B 0,C 180,E1 -20870.144,E2 -20870.144} C_VEL
LIN {X 0,Y 406.016,Z 502.153,A -85,B 0,C 180,E1 -20873.14,E2 -20873.14} C_VEL
LIN {X 0,Y 403.007,Z 496.84,A -85,B 0,C 180,E1 -20880.711,E2 -20880.711} C_VEL
LIN {X 0,Y 403.667,Z 499.483,A -85,B 0,C 180,E1 -20884.831,E2 -20884.831} C_VEL
LIN {X 0,Y 406.05,Z 502.204,A -85,B 0,C 180,E1 -20888.568,E2 -20888.568} C_VEL
LIN {X 0,Y 408.637,Z 506.362,A -85,B 0,C 180,E1 -20891.289,E2 -20891.289} C_VEL
LIN {X 0,Y 409.689,Z 507.854,A -85,B 0,C 180,E1 -20892.188,E2 -20892.188} C_VEL
LIN {X 0,Y 413.229,Z 513.15,A -85,B 0,C 180,E1 -20894.79,E2 -20894.79} C_VEL
LIN {X 0,Y 416.523,Z 518.143,A -85,B 0,C 180,E1 -20896.814,E2 -20896.814} C_VEL
LIN {X 0,Y 419.575,Z 523.022,A -85,B 0,C 180,E1 -20898.479,E2 -20898.479} C_VEL
LIN {X 0,Y 426.109,Z 535.032,A -85,B 0,C 180,E1 -20901.618,E2 -20901.618} C_VEL
LIN {X 0,Y 432.734,Z 548.357,A -85,B 0,C 180,E1 -20904.361,E2 -20904.361} C_VEL
LIN {X 0,Y 415.839,Z 757.029,A -85,B 0,C 180,E1 -20907.719,E2 -20907.719} C_VEL
LIN {X 0,Y 412.084,Z 783.835,A -85,B 0,C 180,E1 -20908.28,E2 -20908.28} C_VEL
LIN {X 0,Y 407.847,Z 805.498,A -85,B 0,C 180,E1 -20908.871,E2 -20908.871} C_VEL
LIN {X 0,Y 401.88,Z 829.898,A -85,B 0,C 180,E1 -20909.736,E2 -20909.736} C_VEL
LIN {X 0,Y 396.158,Z 849.397,A -85,B 0,C 180,E1 -20910.608,E2 -20910.608} C_VEL
LIN {X 0,Y 389.177,Z 870.341,A -85,B 0,C 180,E1 -20911.743,E2 -20911.743} C_VEL
LIN {X 0,Y 380.702,Z 892.427,A -85,B 0,C 180,E1 -20913.226,E2 -20913.226} C_VEL
LIN {X 0,Y 372.817,Z 910.888,A -85,B 0,C 180,E1 -20914.712,E2 -20914.712} C_VEL
LIN {X 0,Y 362.773,Z 932.271,A -85,B 0,C 180,E1 -20916.804,E2 -20916.804} C_VEL
LIN {X 0,Y 354.101,Z 949.195,A -85,B 0,C 180,E1 -20918.799,E2 -20918.799} C_VEL
LIN {X 0,Y 343.991,Z 967.716,A -85,B 0,C 180,E1 -20921.415,E2 -20921.415} C_VEL
LIN {X 0,Y 334.973,Z 983.222,A -85,B 0,C 180,E1 -20924.068,E2 -20924.068} C_VEL
LIN {X 0,Y 325.607,Z 998.873,A -85,B 0,C 180,E1 -20927.261,E2 -20927.261} C_VEL
LIN {X 0,Y 317.11,Z 1012.523,A -85,B 0,C 180,E1 -20930.67,E2 -20930.67} C_VEL
LIN {X 0,Y 309.394,Z 1025.113,A -85,B 0,C 180,E1 -20934.429,E2 -20934.429} C_VEL
LIN {X 0,Y 302.628,Z 1036.239,A -85,B 0,C 180,E1 -20938.531,E2 -20938.531} C_VEL
LIN {X 0,Y 297.469,Z 1045.339,A -85,B 0,C 180,E1 -20942.58,E2 -20942.58} C_VEL
LIN {X 0,Y 293.076,Z 1053.875,A -85,B 0,C 180,E1 -20947.324,E2 -20947.324} C_VEL
LIN {X 0,Y 290.474,Z 1059.872,A -85,B 0,C 180,E1 -20951.537,E2 -20951.537} C_VEL
LIN {X 0,Y 288.747,Z 1065.188,A -85,B 0,C 180,E1 -20956.38,E2 -20956.38} C_VEL
LIN {X 0,Y 288.079,Z 1068.483,A -85,B 0,C 180,E1 -20960.813,E2 -20960.813} C_VEL
LIN {X 0,Y 287.967,Z 1070.282,A -85,B 0,C 180,E1 -20964.621,E2 -20964.621} C_VEL
LIN {X 0,Y 287.985,Z 1071.082,A -85,B 0,C 180,E1 -20968.408,E2 -20968.408} C_VEL
LIN {X 0,Y 287.985,Z 1070.834,A -85,B 0,C 180,E1 -20972.587,E2 -20972.587} C_VEL
LIN {X 0,Y 287.986,Z 1069.107,A -85,B 0,C 180,E1 -20976.98,E2 -20976.98} C_VEL
LIN {X 0,Y 288.257,Z 1066.378,A -85,B 0,C 180,E1 -20980.998,E2 -20980.998} C_VEL
LIN {X 0,Y 289.162,Z 1062.293,A -85,B 0,C 180,E1 -20985.256,E2 -20985.256} C_VEL
LIN {X 0,Y 291.363,Z 1055.687,A -85,B 0,C 180,E1 -20990.28,E2 -20990.28} C_VEL
LIN {X 0,Y 294.375,Z 1048.627,A -85,B 0,C 180,E1 -20994.481,E2 -20994.481} C_VEL
LIN {X 0,Y 299.508,Z 1038.299,A -85,B 0,C 180,E1 -20999.39,E2 -20999.39} C_VEL
LIN {X 0,Y 304.87,Z 1028.398,A -85,B 0,C 180,E1 -21003.21,E2 -21003.21} C_VEL
LIN {X 0,Y 312.45,Z 1015.068,A -85,B 0,C 180,E1 -21007.447,E2 -21007.447} C_VEL
LIN {X 0,Y 319.807,Z 1002.235,A -85,B 0,C 180,E1 -21010.802,E2 -21010.802} C_VEL
LIN {X 0,Y 328.611,Z 986.823,A -85,B 0,C 180,E1 -21014.17,E2 -21014.17} C_VEL
LIN {X 0,Y 337.253,Z 971.088,A -85,B 0,C 180,E1 -21017.007,E2 -21017.007} C_VEL
LIN {X 0,Y 346.72,Z 953.222,A -85,B 0,C 180,E1 -21019.71,E2 -21019.71} C_VEL
LIN {X 0,Y 355.534,Z 935.243,A -85,B 0,C 180,E1 -21021.949,E2 -21021.949} C_VEL
LIN {X 0,Y 364.125,Z 916.576,A -85,B 0,C 180,E1 -21023.914,E2 -21023.914} C_VEL
LIN {X 0,Y 372.799,Z 895.718,A -85,B 0,C 180,E1 -21025.719,E2 -21025.719} C_VEL
LIN {X 0,Y 379.948,Z 876.799,A -85,B 0,C 180,E1 -21027.087,E2 -21027.087} C_VEL
LIN {X 0,Y 387.699,Z 853.539,A -85,B 0,C 180,E1 -21028.471,E2 -21028.471} C_VEL
LIN {X 0,Y 393.582,Z 833.06,A -85,B 0,C 180,E1 -21029.454,E2 -21029.454} C_VEL
LIN {X 0,Y 399.52,Z 808.81,A -85,B 0,C 180,E1 -21030.383,E2 -21030.383} C_VEL
LIN {X 0,Y 403.959,Z 785.801,A -85,B 0,C 180,E1 -21031.049,E2 -21031.049} C_VEL
LIN {X 0,Y 407.539,Z 760.984,A -85,B 0,C 180,E1 -21031.605,E2 -21031.605} C_VEL
LIN {X 0,Y 412.003,Z 705.545,A -85,B 0,C 180,E1 -21032.541,E2 -21032.541} C_VEL
LIN {X 0,Y 424.479,Z 542.553,A -85,B 0,C 180,E1 -21035.21,E2 -21035.21} C_VEL
LIN {X 0,Y 417.996,Z 529.525,A -85,B 0,C 180,E1 -21037.645,E2 -21037.645} C_VEL
LIN {X 0,Y 411.257,Z 516.965,A -85,B 0,C 180,E1 -21040.507,E2 -21040.507} C_VEL
LIN {X 0,Y 407.07,Z 510.274,A -85,B 0,C 180,E1 -21042.488,E2 -21042.488} C_VEL
LIN {X 0,Y 401.903,Z 502.437,A -85,B 0,C 180,E1 -21045.3,E2 -21045.3} C_VEL
LIN {X 0,Y 398.522,Z 497.598,A -85,B 0,C 180,E1 -21047.465,E2 -21047.465} C_VEL
LIN {X 0,Y 395.306,Z 492.897,A -85,B 0,C 180,E1 -21049.949,E2 -21049.949} C_VEL
LIN {X 0,Y 392.528,Z 488.937,A -85,B 0,C 180,E1 -21052.683,E2 -21052.683} C_VEL
LIN {X 0,Y 391.947,Z 487.896,A -85,B 0,C 180,E1 -21053.408,E2 -21053.408} C_VEL
LIN {X 0,Y 388.991,Z 482.499,A -85,B 0,C 180,E1 -21061.326,E2 -21061.326} C_VEL
LIN {X 0,Y 392.262,Z 488.286,A -85,B 0,C 180,E1 -21069.389,E2 -21069.389} C_VEL
LIN {X 0,Y 395.071,Z 492.677,A -85,B 0,C 180,E1 -21072.275,E2 -21072.275} C_VEL
LIN {X 0,Y 396.19,Z 494.16,A -85,B 0,C 180,E1 -21073.203,E2 -21073.203} C_VEL
LIN {X 0,Y 399.81,Z 499.457,A -85,B 0,C 180,E1 -21075.819,E2 -21075.819} C_VEL
LIN {X 0,Y 403.5,Z 504.884,A -85,B 0,C 180,E1 -21078.045,E2 -21078.045} C_VEL
LIN {X 0,Y 408.402,Z 512.099,A -85,B 0,C 180,E1 -21080.569,E2 -21080.569} C_VEL
LIN {X 0,Y 414.685,Z 522.176,A -85,B 0,C 180,E1 -21083.369,E2 -21083.369} C_VEL
LIN {X 0,Y 421.744,Z 533.898,A -85,B 0,C 180,E1 -21086.091,E2 -21086.091} C_VEL
LIN {X 0,Y 424.679,Z 539.346,A -85,B 0,C 180,E1 -21087.141,E2 -21087.141} C_VEL
LIN {X 0,Y 408.507,Z 746.677,A -85,B 0,C 180,E1 -21090.527,E2 -21090.527} C_VEL
LIN {X 0,Y 404.973,Z 773.299,A -85,B 0,C 180,E1 -21091.123,E2 -21091.123} C_VEL
LIN {X 0,Y 401.215,Z 793.937,A -85,B 0,C 180,E1 -21091.742,E2 -21091.742} C_VEL
LIN {X 0,Y 395.957,Z 817.28,A -85,B 0,C 180,E1 -21092.63,E2 -21092.63} C_VEL
LIN {X 0,Y 389.927,Z 839.1,A -85,B 0,C 180,E1 -21093.684,E2 -21093.684} C_VEL
LIN {X 0,Y 382.84,Z 861.502,A -85,B 0,C 180,E1 -21095.004,E2 -21095.004} C_VEL
LIN {X 0,Y 375.101,Z 882.36,A -85,B 0,C 180,E1 -21096.516,E2 -21096.516} C_VEL
LIN {X 0,Y 366.838,Z 902.668,A -85,B 0,C 180,E1 -21098.279,E2 -21098.279} C_VEL
LIN {X 0,Y 358.002,Z 922.016,A -85,B 0,C 180,E1 -21100.317,E2 -21100.317} C_VEL
LIN {X 0,Y 349.622,Z 939.11,A -85,B 0,C 180,E1 -21102.451,E2 -21102.451} C_VEL
LIN {X 0,Y 340.182,Z 957.009,A -85,B 0,C 180,E1 -21105.136,E2 -21105.136} C_VEL
LIN {X 0,Y 331.75,Z 972.148,A -85,B 0,C 180,E1 -21107.855,E2 -21107.855} C_VEL
LIN {X 0,Y 322.237,Z 988.539,A -85,B 0,C 180,E1 -21111.413,E2 -21111.413} C_VEL
LIN {X 0,Y 314.833,Z 1001.002,A -85,B 0,C 180,E1 -21114.689,E2 -21114.689} C_VEL
LIN {X 0,Y 306.895,Z 1014.378,A -85,B 0,C 180,E1 -21118.968,E2 -21118.968} C_VEL
LIN {X 0,Y 301.308,Z 1024.027,A -85,B 0,C 180,E1 -21122.745,E2 -21122.745} C_VEL
LIN {X 0,Y 295.904,Z 1033.979,A -85,B 0,C 180,E1 -21127.552,E2 -21127.552} C_VEL
LIN {X 0,Y 292.592,Z 1040.756,A -85,B 0,C 180,E1 -21131.676,E2 -21131.676} C_VEL
LIN {X 0,Y 290.083,Z 1046.948,A -85,B 0,C 180,E1 -21136.444,E2 -21136.444} C_VEL
LIN {X 0,Y 288.764,Z 1051.05,A -85,B 0,C 180,E1 -21140.835,E2 -21140.835} C_VEL
LIN {X 0,Y 288.211,Z 1053.685,A -85,B 0,C 180,E1 -21144.825,E2 -21144.825} C_VEL
LIN {X 0,Y 288.019,Z 1055.463,A -85,B 0,C 180,E1 -21149.403,E2 -21149.403} C_VEL
LIN {X 0,Y 288.005,Z 1055.705,A -85,B 0,C 180,E1 -21153.782,E2 -21153.782} C_VEL
LIN {X 0,Y 288.123,Z 1054.94,A -85,B 0,C 180,E1 -21157.578,E2 -21157.578} C_VEL
LIN {X 0,Y 288.513,Z 1053.115,A -85,B 0,C 180,E1 -21161.596,E2 -21161.596} C_VEL
LIN {X 0,Y 289.793,Z 1049.283,A -85,B 0,C 180,E1 -21166.641,E2 -21166.641} C_VEL
LIN {X 0,Y 291.925,Z 1044.394,A -85,B 0,C 180,E1 -21171.078,E2 -21171.078} C_VEL
LIN {X 0,Y 295.571,Z 1037.495,A -85,B 0,C 180,E1 -21175.874,E2 -21175.874} C_VEL
LIN {X 0,Y 300.228,Z 1029.43,A -85,B 0,C 180,E1 -21180.192,E2 -21180.192} C_VEL
LIN {X 0,Y 306.254,Z 1019.849,A -85,B 0,C 180,E1 -21184.39,E2 -21184.39} C_VEL
LIN {X 0,Y 313.616,Z 1008.268,A -85,B 0,C 180,E1 -21188.441,E2 -21188.441} C_VEL
LIN {X 0,Y 321.511,Z 996.063,A -85,B 0,C 180,E1 -21191.988,E2 -21191.988} C_VEL
LIN {X 0,Y 330.651,Z 981.473,A -85,B 0,C 180,E1 -21195.447,E2 -21195.447} C_VEL
LIN {X 0,Y 339.237,Z 967.4,A -85,B 0,C 180,E1 -21198.231,E2 -21198.231} C_VEL
LIN {X 0,Y 349.394,Z 949.786,A -85,B 0,C 180,E1 -21201.115,E2 -21201.115} C_VEL
LIN {X 0,Y 358.057,Z 933.776,A -85,B 0,C 180,E1 -21203.301,E2 -21203.301} C_VEL
LIN {X 0,Y 368.287,Z 913.322,A -85,B 0,C 180,E1 -21205.624,E2 -21205.624} C_VEL
LIN {X 0,Y 376.198,Z 895.916,A -85,B 0,C 180,E1 -21207.269,E2 -21207.269} C_VEL
LIN {X 0,Y 384.849,Z 875.072,A -85,B 0,C 180,E1 -21208.926,E2 -21208.926} C_VEL
LIN {X 0,Y 392.189,Z 854.792,A -85,B 0,C 180,E1 -21210.245,E2 -21210.245} C_VEL
LIN {X 0,Y 398.983,Z 833.545,A -85,B 0,C 180,E1 -21211.402,E2 -21211.402} C_VEL
LIN {X 0,Y 405.258,Z 810.118,A -85,B 0,C 180,E1 -21212.421,E2 -21212.421} C_VEL
LIN {X 0,Y 410.097,Z 788.311,A -85,B 0,C 180,E1 -21213.173,E2 -21213.173} C_VEL
LIN {X 0,Y 414.512,Z 762.333,A -85,B 0,C 180,E1 -21213.85,E2 -21213.85} C_VEL
LIN {X 0,Y 416.266,Z 748.791,A -85,B 0,C 180,E1 -21214.126,E2 -21214.126} C_VEL
LIN {X 0,Y 416.563,Z 741.256,A -85,B 0,C 180,E1 -21214.383,E2 -21214.383} C_VEL
LIN {X 0,Y 415.521,Z 721.593,A -85,B 0,C 180,E1 -21215.481,E2 -21215.481} C_VEL
LIN {X 0,Y 415.705,Z 715.097,A -85,B 0,C 180,E1 -21215.681,E2 -21215.681} C_VEL
LIN {X 0,Y 429.308,Z 549.524,A -85,B 0,C 180,E1 -21218.326,E2 -21218.326} C_VEL
LIN {X 0,Y 423.035,Z 538.788,A -85,B 0,C 180,E1 -21220.987,E2 -21220.987} C_VEL
LIN {X 0,Y 417.915,Z 530.42,A -85,B 0,C 180,E1 -21223.494,E2 -21223.494} C_VEL
LIN {X 0,Y 413.316,Z 523.144,A -85,B 0,C 180,E1 -21226.143,E2 -21226.143} C_VEL
LIN {X 0,Y 410.314,Z 518.541,A -85,B 0,C 180,E1 -21228.188,E2 -21228.188} C_VEL
LIN {X 0,Y 407.612,Z 514.346,A -85,B 0,C 180,E1 -21230.398,E2 -21230.398} C_VEL
LIN {X 0,Y 404.535,Z 509.534,A -85,B 0,C 180,E1 -21233.756,E2 -21233.756} C_VEL
LIN {X 0,Y 402.031,Z 504.781,A -85,B 0,C 180,E1 -21240.855,E2 -21240.855} C_VEL
LIN {X 0,Y 404.899,Z 510.028,A -85,B 0,C 180,E1 -21248.378,E2 -21248.378} C_VEL
LIN {X 0,Y 407.506,Z 514.248,A -85,B 0,C 180,E1 -21251.177,E2 -21251.177} C_VEL
LIN {X 0,Y 409.195,Z 517.002,A -85,B 0,C 180,E1 -21252.633,E2 -21252.633} C_VEL
LIN {X 0,Y 411.637,Z 520.527,A -85,B 0,C 180,E1 -21254.417,E2 -21254.417} C_VEL
LIN {X 0,Y 415.064,Z 525.883,A -85,B 0,C 180,E1 -21256.587,E2 -21256.587} C_VEL
LIN {X 0,Y 417.873,Z 530.518,A -85,B 0,C 180,E1 -21258.16,E2 -21258.16} C_VEL
LIN {X 0,Y 423.983,Z 542.072,A -85,B 0,C 180,E1 -21261.187,E2 -21261.187} C_VEL
LIN {X 0,Y 429.212,Z 552.824,A -85,B 0,C 180,E1 -21263.45,E2 -21263.45} C_VEL
LIN {X 0,Y 412.278,Z 756.881,A -85,B 0,C 180,E1 -21266.724,E2 -21266.724} C_VEL
LIN {X 0,Y 408.476,Z 783.53,A -85,B 0,C 180,E1 -21267.277,E2 -21267.277} C_VEL
LIN {X 0,Y 404.178,Z 805.123,A -85,B 0,C 180,E1 -21267.859,E2 -21267.859} C_VEL
LIN {X 0,Y 397.959,Z 830.029,A -85,B 0,C 180,E1 -21268.732,E2 -21268.732} C_VEL
LIN {X 0,Y 392.12,Z 849.486,A -85,B 0,C 180,E1 -21269.595,E2 -21269.595} C_VEL
LIN {X 0,Y 384.643,Z 871.4,A -85,B 0,C 180,E1 -21270.779,E2 -21270.779} C_VEL
LIN {X 0,Y 375.982,Z 893.24,A -85,B 0,C 180,E1 -21272.254,E2 -21272.254} C_VEL
LIN {X 0,Y 367.268,Z 913.073,A -85,B 0,C 180,E1 -21273.864,E2 -21273.864} C_VEL
LIN {X 0,Y 357.356,Z 933.354,A -85,B 0,C 180,E1 -21275.883,E2 -21275.883} C_VEL
LIN {X 0,Y 348.137,Z 950.795,A -85,B 0,C 180,E1 -21277.964,E2 -21277.964} C_VEL
LIN {X 0,Y 337.465,Z 969.534,A -85,B 0,C 180,E1 -21280.681,E2 -21280.681} C_VEL
LIN {X 0,Y 328.891,Z 983.777,A -85,B 0,C 180,E1 -21283.161,E2 -21283.161} C_VEL
LIN {X 0,Y 319.119,Z 999.452,A -85,B 0,C 180,E1 -21286.423,E2 -21286.423} C_VEL
LIN {X 0,Y 310.753,Z 1012.387,A -85,B 0,C 180,E1 -21289.703,E2 -21289.703} C_VEL
LIN {X 0,Y 302.691,Z 1024.969,A -85,B 0,C 180,E1 -21293.516,E2 -21293.516} C_VEL
LIN {X 0,Y 295.454,Z 1036.304,A -85,B 0,C 180,E1 -21297.786,E2 -21297.786} C_VEL
LIN {X 0,Y 289.701,Z 1045.994,A -85,B 0,C 180,E1 -21302.228,E2 -21302.228} C_VEL
LIN {X 0,Y 285.17,Z 1054.313,A -85,B 0,C 180,E1 -21307.095,E2 -21307.095} C_VEL
LIN {X 0,Y 282.411,Z 1060.425,A -85,B 0,C 180,E1 -21311.599,E2 -21311.599} C_VEL
LIN {X 0,Y 280.642,Z 1065.65,A -85,B 0,C 180,E1 -21316.819,E2 -21316.819} C_VEL
LIN {X 0,Y 280.071,Z 1068.517,A -85,B 0,C 180,E1 -21320.962,E2 -21320.962} C_VEL
LIN {X 0,Y 279.968,Z 1070.217,A -85,B 0,C 180,E1 -21324.877,E2 -21324.877} C_VEL
LIN {X 0,Y 279.997,Z 1070.97,A -85,B 0,C 180,E1 -21329.217,E2 -21329.217} C_VEL
LIN {X 0,Y 279.979,Z 1070.365,A -85,B 0,C 180,E1 -21333.481,E2 -21333.481} C_VEL
LIN {X 0,Y 280.001,Z 1068.643,A -85,B 0,C 180,E1 -21337.593,E2 -21337.593} C_VEL
LIN {X 0,Y 280.361,Z 1065.813,A -85,B 0,C 180,E1 -21341.729,E2 -21341.729} C_VEL
LIN {X 0,Y 281.638,Z 1060.925,A -85,B 0,C 180,E1 -21346.713,E2 -21346.713} C_VEL
LIN {X 0,Y 283.905,Z 1054.806,A -85,B 0,C 180,E1 -21351.27,E2 -21351.27} C_VEL
LIN {X 0,Y 287.616,Z 1046.913,A -85,B 0,C 180,E1 -21355.979,E2 -21355.979} C_VEL
LIN {X 0,Y 292.82,Z 1037.08,A -85,B 0,C 180,E1 -21360.583,E2 -21360.583} C_VEL
LIN {X 0,Y 298.908,Z 1026.533,A -85,B 0,C 180,E1 -21364.658,E2 -21364.658} C_VEL
LIN {X 0,Y 306.651,Z 1013.468,A -85,B 0,C 180,E1 -21368.759,E2 -21368.759} C_VEL
LIN {X 0,Y 314.436,Z 1000.495,A -85,B 0,C 180,E1 -21372.142,E2 -21372.142} C_VEL
LIN {X 0,Y 323.692,Z 984.772,A -85,B 0,C 180,E1 -21375.525,E2 -21375.525} C_VEL
LIN {X 0,Y 331.827,Z 970.468,A -85,B 0,C 180,E1 -21378.097,E2 -21378.097} C_VEL
LIN {X 0,Y 341.415,Z 952.907,A -85,B 0,C 180,E1 -21380.758,E2 -21380.758} C_VEL
LIN {X 0,Y 350.523,Z 934.858,A -85,B 0,C 180,E1 -21383.008,E2 -21383.008} C_VEL
LIN {X 0,Y 359.801,Z 915.22,A -85,B 0,C 180,E1 -21385.065,E2 -21385.065} C_VEL
LIN {X 0,Y 368.539,Z 894.582,A -85,B 0,C 180,E1 -21386.824,E2 -21386.824} C_VEL
LIN {X 0,Y 376.276,Z 874.492,A -85,B 0,C 180,E1 -21388.254,E2 -21388.254} C_VEL
LIN {X 0,Y 383.865,Z 851.878,A -85,B 0,C 180,E1 -21389.563,E2 -21389.563} C_VEL
LIN {X 0,Y 389.528,Z 832.498,A -85,B 0,C 180,E1 -21390.48,E2 -21390.48} C_VEL
LIN {X 0,Y 395.621,Z 807.974,A -85,B 0,C 180,E1 -21391.406,E2 -21391.406} C_VEL
LIN {X 0,Y 400.052,Z 785.373,A -85,B 0,C 180,E1 -21392.052,E2 -21392.052} C_VEL
LIN {X 0,Y 403.701,Z 760.378,A -85,B 0,C 180,E1 -21392.605,E2 -21392.605} C_VEL
LIN {X 0,Y 408.476,Z 702.307,A -85,B 0,C 180,E1 -21393.582,E2 -21393.582} C_VEL
LIN {X 0,Y 420.683,Z 546.685,A -85,B 0,C 180,E1 -21396.13,E2 -21396.13} C_VEL
LIN {X 0,Y 413.283,Z 531.787,A -85,B 0,C 180,E1 -21399.092,E2 -21399.092} C_VEL
LIN {X 0,Y 407.708,Z 521.486,A -85,B 0,C 180,E1 -21401.638,E2 -21401.638} C_VEL
LIN {X 0,Y 402.69,Z 513.685,A -85,B 0,C 180,E1 -21404.223,E2 -21404.223} C_VEL
LIN {X 0,Y 399.532,Z 508.91,A -85,B 0,C 180,E1 -21406.098,E2 -21406.098} C_VEL
LIN {X 0,Y 397.13,Z 505.283,A -85,B 0,C 180,E1 -21407.716,E2 -21407.716} C_VEL
LIN {X 0,Y 393.987,Z 500.614,A -85,B 0,C 180,E1 -21410.21,E2 -21410.21} C_VEL
LIN {X 0,Y 391.246,Z 496.487,A -85,B 0,C 180,E1 -21413.027,E2 -21413.027} C_VEL
LIN {X 0,Y 390.728,Z 495.704,A -85,B 0,C 180,E1 -21413.682,E2 -21413.682} C_VEL
LIN {X 0,Y 388.012,Z 490.465,A -85,B 0,C 180,E1 -21421.329,E2 -21421.329} C_VEL
LIN {X 0,Y 391.156,Z 496.248,A -85,B 0,C 180,E1 -21429.268,E2 -21429.268} C_VEL
LIN {X 0,Y 394.104,Z 500.734,A -85,B 0,C 180,E1 -21432.305,E2 -21432.305} C_VEL
LIN {X 0,Y 398.294,Z 507.008,A -85,B 0,C 180,E1 -21435.507,E2 -21435.507} C_VEL
LIN {X 0,Y 401.9,Z 512.442,A -85,B 0,C 180,E1 -21437.744,E2 -21437.744} C_VEL
LIN {X 0,Y 406.635,Z 519.608,A -85,B 0,C 180,E1 -21440.249,E2 -21440.249} C_VEL
LIN {X 0,Y 412.649,Z 529.458,A -85,B 0,C 180,E1 -21443,E2 -21443} C_VEL
LIN {X 0,Y 419.569,Z 541.223,A -85,B 0,C 180,E1 -21445.739,E2 -21445.739} C_VEL
LIN {X 0,Y 420.876,Z 543.854,A -85,B 0,C 180,E1 -21446.231,E2 -21446.231} C_VEL
LIN {X 0,Y 404.626,Z 746.959,A -85,B 0,C 180,E1 -21449.542,E2 -21449.542} C_VEL
LIN {X 0,Y 401.028,Z 773.491,A -85,B 0,C 180,E1 -21450.132,E2 -21450.132} C_VEL
LIN {X 0,Y 397.201,Z 794.082,A -85,B 0,C 180,E1 -21450.745,E2 -21450.745} C_VEL
LIN {X 0,Y 391.709,Z 817.882,A -85,B 0,C 180,E1 -21451.646,E2 -21451.646} C_VEL
LIN {X 0,Y 385.55,Z 839.656,A -85,B 0,C 180,E1 -21452.695,E2 -21452.695} C_VEL
LIN {X 0,Y 378.278,Z 862.046,A -85,B 0,C 180,E1 -21454.013,E2 -21454.013} C_VEL
LIN {X 0,Y 370.377,Z 882.821,A -85,B 0,C 180,E1 -21455.517,E2 -21455.517} C_VEL
LIN {X 0,Y 361.905,Z 903.106,A -85,B 0,C 180,E1 -21457.279,E2 -21457.279} C_VEL
LIN {X 0,Y 352.831,Z 922.417,A -85,B 0,C 180,E1 -21459.317,E2 -21459.317} C_VEL
LIN {X 0,Y 344.041,Z 939.832,A -85,B 0,C 180,E1 -21461.502,E2 -21461.502} C_VEL
LIN {X 0,Y 334.478,Z 957.369,A -85,B 0,C 180,E1 -21464.155,E2 -21464.155} C_VEL
LIN {X 0,Y 325.941,Z 972.191,A -85,B 0,C 180,E1 -21466.835,E2 -21466.835} C_VEL
LIN {X 0,Y 316.347,Z 988.176,A -85,B 0,C 180,E1 -21470.322,E2 -21470.322} C_VEL
LIN {X 0,Y 308.595,Z 1000.694,A -85,B 0,C 180,E1 -21473.634,E2 -21473.634} C_VEL
LIN {X 0,Y 300.833,Z 1013.275,A -85,B 0,C 180,E1 -21477.648,E2 -21477.648} C_VEL
LIN {X 0,Y 294.611,Z 1023.418,A -85,B 0,C 180,E1 -21481.631,E2 -21481.631} C_VEL
LIN {X 0,Y 289.198,Z 1032.87,A -85,B 0,C 180,E1 -21486.139,E2 -21486.139} C_VEL
LIN {X 0,Y 285.183,Z 1040.428,A -85,B 0,C 180,E1 -21490.757,E2 -21490.757} C_VEL
LIN {X 0,Y 282.487,Z 1046.527,A -85,B 0,C 180,E1 -21495.445,E2 -21495.445} C_VEL
LIN {X 0,Y 280.863,Z 1051.135,A -85,B 0,C 180,E1 -21500.368,E2 -21500.368} C_VEL
LIN {X 0,Y 280.246,Z 1053.806,A -85,B 0,C 180,E1 -21504.472,E2 -21504.472} C_VEL
LIN {X 0,Y 280.034,Z 1055.508,A -85,B 0,C 180,E1 -21508.785,E2 -21508.785} C_VEL
LIN {X 0,Y 280.003,Z 1055.98,A -85,B 0,C 180,E1 -21513.275,E2 -21513.275} C_VEL
LIN {X 0,Y 280.119,Z 1055.275,A -85,B 0,C 180,E1 -21517.383,E2 -21517.383} C_VEL
LIN {X 0,Y 280.485,Z 1053.606,A -85,B 0,C 180,E1 -21521.38,E2 -21521.38} C_VEL
LIN {X 0,Y 281.592,Z 1050.422,A -85,B 0,C 180,E1 -21526.079,E2 -21526.079} C_VEL
LIN {X 0,Y 283.879,Z 1045.321,A -85,B 0,C 180,E1 -21531.055,E2 -21531.055} C_VEL
LIN {X 0,Y 287.209,Z 1039.23,A -85,B 0,C 180,E1 -21535.575,E2 -21535.575} C_VEL
LIN {X 0,Y 292.452,Z 1030.6,A -85,B 0,C 180,E1 -21540.504,E2 -21540.504} C_VEL
LIN {X 0,Y 298.182,Z 1021.813,A -85,B 0,C 180,E1 -21544.521,E2 -21544.521} C_VEL
LIN {X 0,Y 306.424,Z 1009.502,A -85,B 0,C 180,E1 -21549.048,E2 -21549.048} C_VEL
LIN {X 0,Y 314.05,Z 998.143,A -85,B 0,C 180,E1 -21552.452,E2 -21552.452} C_VEL
LIN {X 0,Y 324.098,Z 982.835,A -85,B 0,C 180,E1 -21556.214,E2 -21556.214} C_VEL
LIN {X 0,Y 332.708,Z 969.207,A -85,B 0,C 180,E1 -21558.967,E2 -21558.967} C_VEL
LIN {X 0,Y 343.144,Z 951.871,A -85,B 0,C 180,E1 -21561.883,E2 -21561.883} C_VEL
LIN {X 0,Y 352.231,Z 935.616,A -85,B 0,C 180,E1 -21564.141,E2 -21564.141} C_VEL
LIN {X 0,Y 361.829,Z 917.319,A -85,B 0,C 180,E1 -21566.283,E2 -21566.283} C_VEL
LIN {X 0,Y 370.857,Z 898.112,A -85,B 0,C 180,E1 -21568.135,E2 -21568.135} C_VEL
LIN {X 0,Y 378.885,Z 879.443,A -85,B 0,C 180,E1 -21569.651,E2 -21569.651} C_VEL
LIN {X 0,Y 387.606,Z 856.479,A -85,B 0,C 180,E1 -21571.18,E2 -21571.18} C_VEL
LIN {X 0,Y 394.201,Z 836.465,A -85,B 0,C 180,E1 -21572.281,E2 -21572.281} C_VEL
LIN {X 0,Y 401.217,Z 811.37,A -85,B 0,C 180,E1 -21573.387,E2 -21573.387} C_VEL
LIN {X 0,Y 406.128,Z 789.851,A -85,B 0,C 180,E1 -21574.13,E2 -21574.13} C_VEL
LIN {X 0,Y 410.704,Z 764.047,A -85,B 0,C 180,E1 -21574.81,E2 -21574.81} C_VEL
LIN {X 0,Y 413.436,Z 741.716,A -85,B 0,C 180,E1 -21575.245,E2 -21575.245} C_VEL
LIN {X 0,Y 415.705,Z 715.097,A -85,B 0,C 180,E1 -21575.681,E2 -21575.681} C_VEL
LIN {X 0,Y 415.888,Z 707.543,A -85,B 0,C 180,E1 -21575.929,E2 -21575.929} C_VEL
LIN {X 0,Y 414.926,Z 687.871,A -85,B 0,C 180,E1 -21577.027,E2 -21577.027} C_VEL
LIN {X 0,Y 415.159,Z 681.376,A -85,B 0,C 180,E1 -21577.228,E2 -21577.228} C_VEL
LIN {X 0,Y 425.901,Z 554.4,A -85,B 0,C 180,E1 -21579.237,E2 -21579.237} C_VEL
LIN {X 0,Y 419.442,Z 543.145,A -85,B 0,C 180,E1 -21582.162,E2 -21582.162} C_VEL
LIN {X 0,Y 414.203,Z 534.559,A -85,B 0,C 180,E1 -21584.959,E2 -21584.959} C_VEL
LIN {X 0,Y 410.956,Z 529.462,A -85,B 0,C 180,E1 -21586.993,E2 -21586.993} C_VEL
LIN {X 0,Y 408.862,Z 526.106,A -85,B 0,C 180,E1 -21588.503,E2 -21588.503} C_VEL
LIN {X 0,Y 406.319,Z 522.059,A -85,B 0,C 180,E1 -21590.653,E2 -21590.653} C_VEL
LIN {X 0,Y 403.45,Z 517.419,A -85,B 0,C 180,E1 -21593.882,E2 -21593.882} C_VEL
LIN {X 0,Y 401.055,Z 512.724,A -85,B 0,C 180,E1 -21600.857,E2 -21600.857} C_VEL
LIN {X 0,Y 403.802,Z 517.98,A -85,B 0,C 180,E1 -21608.257,E2 -21608.257} C_VEL
LIN {X 0,Y 406.377,Z 522.134,A -85,B 0,C 180,E1 -21611.065,E2 -21611.065} C_VEL
LIN {X 0,Y 410.252,Z 528.245,A -85,B 0,C 180,E1 -21614.179,E2 -21614.179} C_VEL
LIN {X 0,Y 413.501,Z 533.436,A -85,B 0,C 180,E1 -21616.29,E2 -21616.29} C_VEL
LIN {X 0,Y 416.125,Z 537.897,A -85,B 0,C 180,E1 -21617.804,E2 -21617.804} C_VEL
LIN {X 0,Y 421.95,Z 549.263,A -85,B 0,C 180,E1 -21620.785,E2 -21620.785} C_VEL
LIN {X 0,Y 425.774,Z 557.6,A -85,B 0,C 180,E1 -21622.529,E2 -21622.529} C_VEL
LIN {X 0,Y 408.854,Z 756.627,A -85,B 0,C 180,E1 -21625.709,E2 -21625.709} C_VEL
LIN {X 0,Y 404.961,Z 783.408,A -85,B 0,C 180,E1 -21626.26,E2 -21626.26} C_VEL
LIN {X 0,Y 400.596,Z 804.942,A -85,B 0,C 180,E1 -21626.833,E2 -21626.833} C_VEL
LIN {X 0,Y 394.541,Z 828.877,A -85,B 0,C 180,E1 -21627.657,E2 -21627.657} C_VEL
LIN {X 0,Y 388.207,Z 849.575,A -85,B 0,C 180,E1 -21628.562,E2 -21628.562} C_VEL
LIN {X 0,Y 380.573,Z 871.453,A -85,B 0,C 180,E1 -21629.735,E2 -21629.735} C_VEL
LIN {X 0,Y 371.72,Z 893.243,A -85,B 0,C 180,E1 -21631.197,E2 -21631.197} C_VEL
LIN {X 0,Y 362.466,Z 913.79,A -85,B 0,C 180,E1 -21632.861,E2 -21632.861} C_VEL
LIN {X 0,Y 352.59,Z 933.381,A -85,B 0,C 180,E1 -21634.817,E2 -21634.817} C_VEL
LIN {X 0,Y 342.856,Z 951.283,A -85,B 0,C 180,E1 -21636.958,E2 -21636.958} C_VEL
LIN {X 0,Y 332.195,Z 969.387,A -85,B 0,C 180,E1 -21639.597,E2 -21639.597} C_VEL
LIN {X 0,Y 322.814,Z 984.464,A -85,B 0,C 180,E1 -21642.245,E2 -21642.245} C_VEL
LIN {X 0,Y 312.22,Z 1000.737,A -85,B 0,C 180,E1 -21645.721,E2 -21645.721} C_VEL
LIN {X 0,Y 303.63,Z 1013.532,A -85,B 0,C 180,E1 -21649.055,E2 -21649.055} C_VEL
LIN {X 0,Y 294.606,Z 1026.928,A -85,B 0,C 180,E1 -21653.32,E2 -21653.32} C_VEL
LIN {X 0,Y 288.02,Z 1036.849,A -85,B 0,C 180,E1 -21657.209,E2 -21657.209} C_VEL
LIN {X 0,Y 281.941,Z 1046.596,A -85,B 0,C 180,E1 -21661.857,E2 -21661.857} C_VEL
LIN {X 0,Y 277.43,Z 1054.442,A -85,B 0,C 180,E1 -21666.643,E2 -21666.643} C_VEL
LIN {X 0,Y 274.416,Z 1060.8,A -85,B 0,C 180,E1 -21671.518,E2 -21671.518} C_VEL
LIN {X 0,Y 272.672,Z 1065.618,A -85,B 0,C 180,E1 -21676.643,E2 -21676.643} C_VEL
LIN {X 0,Y 272.073,Z 1068.433,A -85,B 0,C 180,E1 -21680.908,E2 -21680.908} C_VEL
LIN {X 0,Y 271.968,Z 1070.223,A -85,B 0,C 180,E1 -21685.361,E2 -21685.361} C_VEL
LIN {X 0,Y 272.005,Z 1070.724,A -85,B 0,C 180,E1 -21689.789,E2 -21689.789} C_VEL
LIN {X 0,Y 271.975,Z 1070.003,A -85,B 0,C 180,E1 -21694.005,E2 -21694.005} C_VEL
LIN {X 0,Y 272.005,Z 1068.413,A -85,B 0,C 180,E1 -21697.817,E2 -21697.817} C_VEL
LIN {X 0,Y 272.412,Z 1065.575,A -85,B 0,C 180,E1 -21702.077,E2 -21702.077} C_VEL
LIN {X 0,Y 273.802,Z 1060.673,A -85,B 0,C 180,E1 -21707.206,E2 -21707.206} C_VEL
LIN {X 0,Y 276.24,Z 1054.546,A -85,B 0,C 180,E1 -21711.89,E2 -21711.89} C_VEL
LIN {X 0,Y 280.198,Z 1046.645,A -85,B 0,C 180,E1 -21716.72,E2 -21716.72} C_VEL
LIN {X 0,Y 285.703,Z 1036.797,A -85,B 0,C 180,E1 -21721.43,E2 -21721.43} C_VEL
LIN {X 0,Y 292.115,Z 1026.242,A -85,B 0,C 180,E1 -21725.584,E2 -21725.584} C_VEL
LIN {X 0,Y 300.214,Z 1013.16,A -85,B 0,C 180,E1 -21729.753,E2 -21729.753} C_VEL
LIN {X 0,Y 308.335,Z 1000.179,A -85,B 0,C 180,E1 -21733.176,E2 -21733.176} C_VEL
LIN {X 0,Y 317.943,Z 984.437,A -85,B 0,C 180,E1 -21736.591,E2 -21736.591} C_VEL
LIN {X 0,Y 326.365,Z 970.121,A -85,B 0,C 180,E1 -21739.177,E2 -21739.177} C_VEL
LIN {X 0,Y 336.576,Z 951.917,A -85,B 0,C 180,E1 -21741.929,E2 -21741.929} C_VEL
LIN {X 0,Y 345.635,Z 934.474,A -85,B 0,C 180,E1 -21744.097,E2 -21744.097} C_VEL
LIN {X 0,Y 355.169,Z 914.815,A -85,B 0,C 180,E1 -21746.15,E2 -21746.15} C_VEL
LIN {X 0,Y 364.176,Z 894.039,A -85,B 0,C 180,E1 -21747.909,E2 -21747.909} C_VEL
LIN {X 0,Y 372.39,Z 873.151,A -85,B 0,C 180,E1 -21749.38,E2 -21749.38} C_VEL
LIN {X 0,Y 379.814,Z 851.354,A -85,B 0,C 180,E1 -21750.62,E2 -21750.62} C_VEL
LIN {X 0,Y 385.604,Z 831.934,A -85,B 0,C 180,E1 -21751.527,E2 -21751.527} C_VEL
LIN {X 0,Y 391.89,Z 806.962,A -85,B 0,C 180,E1 -21752.453,E2 -21752.453} C_VEL
LIN {X 0,Y 396.291,Z 784.838,A -85,B 0,C 180,E1 -21753.076,E2 -21753.076} C_VEL
LIN {X 0,Y 399.998,Z 759.664,A -85,B 0,C 180,E1 -21753.627,E2 -21753.627} C_VEL
LIN {X 0,Y 405.25,Z 696.996,A -85,B 0,C 180,E1 -21754.675,E2 -21754.675} C_VEL
LIN {X 0,Y 417.039,Z 551.019,A -85,B 0,C 180,E1 -21757.046,E2 -21757.046} C_VEL
LIN {X 0,Y 410.551,Z 537.832,A -85,B 0,C 180,E1 -21759.767,E2 -21759.767} C_VEL
LIN {X 0,Y 405.662,Z 528.531,A -85,B 0,C 180,E1 -21762.092,E2 -21762.092} C_VEL
LIN {X 0,Y 400.833,Z 520.865,A -85,B 0,C 180,E1 -21764.667,E2 -21764.667} C_VEL
LIN {X 0,Y 397.667,Z 515.967,A -85,B 0,C 180,E1 -21766.625,E2 -21766.625} C_VEL
LIN {X 0,Y 395.548,Z 512.727,A -85,B 0,C 180,E1 -21768.111,E2 -21768.111} C_VEL
LIN {X 0,Y 392.677,Z 508.329,A -85,B 0,C 180,E1 -21770.473,E2 -21770.473} C_VEL
LIN {X 0,Y 390.029,Z 504.17,A -85,B 0,C 180,E1 -21773.301,E2 -21773.301} C_VEL
LIN {X 0,Y 387.041,Z 498.372,A -85,B 0,C 180,E1 -21781.192,E2 -21781.192} C_VEL
LIN {X 0,Y 390,Z 504.074,A -85,B 0,C 180,E1 -21789.072,E2 -21789.072} C_VEL
LIN {X 0,Y 392.797,Z 508.455,A -85,B 0,C 180,E1 -21792.048,E2 -21792.048} C_VEL
LIN {X 0,Y 396.79,Z 514.56,A -85,B 0,C 180,E1 -21795.193,E2 -21795.193} C_VEL
LIN {X 0,Y 400.43,Z 520.187,A -85,B 0,C 180,E1 -21797.511,E2 -21797.511} C_VEL
LIN {X 0,Y 404.947,Z 527.232,A -85,B 0,C 180,E1 -21799.96,E2 -21799.96} C_VEL
LIN {X 0,Y 410.799,Z 537.02,A -85,B 0,C 180,E1 -21802.701,E2 -21802.701} C_VEL
LIN {X 0,Y 417.195,Z 548.17,A -85,B 0,C 180,E1 -21805.302,E2 -21805.302} C_VEL
LIN {X 0,Y 400.877,Z 747.136,A -85,B 0,C 180,E1 -21808.535,E2 -21808.535} C_VEL
LIN {X 0,Y 397.205,Z 773.682,A -85,B 0,C 180,E1 -21809.122,E2 -21809.122} C_VEL
LIN {X 0,Y 393.285,Z 794.342,A -85,B 0,C 180,E1 -21809.732,E2 -21809.732} C_VEL
LIN {X 0,Y 387.58,Z 818.48,A -85,B 0,C 180,E1 -21810.642,E2 -21810.642} C_VEL
LIN {X 0,Y 381.633,Z 839.09,A -85,B 0,C 180,E1 -21811.624,E2 -21811.624} C_VEL
LIN {X 0,Y 374.467,Z 860.832,A -85,B 0,C 180,E1 -21812.885,E2 -21812.885} C_VEL
LIN {X 0,Y 366.098,Z 882.48,A -85,B 0,C 180,E1 -21814.429,E2 -21814.429} C_VEL
LIN {X 0,Y 357.715,Z 902.093,A -85,B 0,C 180,E1 -21816.117,E2 -21816.117} C_VEL
LIN {X 0,Y 348.074,Z 922.218,A -85,B 0,C 180,E1 -21818.218,E2 -21818.218} C_VEL
LIN {X 0,Y 339.196,Z 939.334,A -85,B 0,C 180,E1 -21820.358,E2 -21820.358} C_VEL
LIN {X 0,Y 328.874,Z 957.728,A -85,B 0,C 180,E1 -21823.14,E2 -21823.14} C_VEL
LIN {X 0,Y 320.057,Z 972.539,A -85,B 0,C 180,E1 -21825.839,E2 -21825.839} C_VEL
LIN {X 0,Y 310.124,Z 988.502,A -85,B 0,C 180,E1 -21829.362,E2 -21829.362} C_VEL
LIN {X 0,Y 302.469,Z 1000.386,A -85,B 0,C 180,E1 -21832.536,E2 -21832.536} C_VEL
LIN {X 0,Y 294.314,Z 1013.068,A -85,B 0,C 180,E1 -21836.608,E2 -21836.608} C_VEL
LIN {X 0,Y 287.583,Z 1023.513,A -85,B 0,C 180,E1 -21840.774,E2 -21840.774} C_VEL
LIN {X 0,Y 281.991,Z 1032.783,A -85,B 0,C 180,E1 -21845.266,E2 -21845.266} C_VEL
LIN {X 0,Y 277.652,Z 1040.456,A -85,B 0,C 180,E1 -21850.039,E2 -21850.039} C_VEL
LIN {X 0,Y 274.859,Z 1046.286,A -85,B 0,C 180,E1 -21854.6,E2 -21854.6} C_VEL
LIN {X 0,Y 272.983,Z 1051.219,A -85,B 0,C 180,E1 -21859.874,E2 -21859.874} C_VEL
LIN {X 0,Y 272.285,Z 1053.927,A -85,B 0,C 180,E1 -21864.098,E2 -21864.098} C_VEL
LIN {X 0,Y 272.046,Z 1055.594,A -85,B 0,C 180,E1 -21868.315,E2 -21868.315} C_VEL
LIN {X 0,Y 272.003,Z 1056.234,A -85,B 0,C 180,E1 -21872.95,E2 -21872.95} C_VEL
LIN {X 0,Y 272.124,Z 1055.545,A -85,B 0,C 180,E1 -21877.389,E2 -21877.389} C_VEL
LIN {X 0,Y 272.518,Z 1053.875,A -85,B 0,C 180,E1 -21881.578,E2 -21881.578} C_VEL
LIN {X 0,Y 273.601,Z 1050.926,A -85,B 0,C 180,E1 -21886.126,E2 -21886.126} C_VEL
LIN {X 0,Y 276.088,Z 1045.75,A -85,B 0,C 180,E1 -21891.456,E2 -21891.456} C_VEL
LIN {X 0,Y 279.397,Z 1039.998,A -85,B 0,C 180,E1 -21895.888,E2 -21895.888} C_VEL
LIN {X 0,Y 285.094,Z 1031.139,A -85,B 0,C 180,E1 -21901.155,E2 -21901.155} C_VEL
LIN {X 0,Y 291.056,Z 1022.416,A -85,B 0,C 180,E1 -21905.25,E2 -21905.25} C_VEL
LIN {X 0,Y 299.612,Z 1010.235,A -85,B 0,C 180,E1 -21909.848,E2 -21909.848} C_VEL
LIN {X 0,Y 307.537,Z 998.894,A -85,B 0,C 180,E1 -21913.316,E2 -21913.316} C_VEL
LIN {X 0,Y 317.43,Z 984.468,A -85,B 0,C 180,E1 -21916.953,E2 -21916.953} C_VEL
LIN {X 0,Y 326.803,Z 970.137,A -85,B 0,C 180,E1 -21919.898,E2 -21919.898} C_VEL
LIN {X 0,Y 336.958,Z 953.954,A -85,B 0,C 180,E1 -21922.68,E2 -21922.68} C_VEL
LIN {X 0,Y 346.802,Z 936.885,A -85,B 0,C 180,E1 -21925.082,E2 -21925.082} C_VEL
LIN {X 0,Y 356.043,Z 919.785,A -85,B 0,C 180,E1 -21927.108,E2 -21927.108} C_VEL
LIN {X 0,Y 365.943,Z 899.567,A -85,B 0,C 180,E1 -21929.09,E2 -21929.09} C_VEL
LIN {X 0,Y 374.138,Z 881.037,A -85,B 0,C 180,E1 -21930.603,E2 -21930.603} C_VEL
LIN {X 0,Y 383.305,Z 857.667,A -85,B 0,C 180,E1 -21932.167,E2 -21932.167} C_VEL
LIN {X 0,Y 390.133,Z 837.471,A -85,B 0,C 180,E1 -21933.276,E2 -21933.276} C_VEL
LIN {X 0,Y 397.109,Z 813.363,A -85,B 0,C 180,E1 -21934.345,E2 -21934.345} C_VEL
LIN {X 0,Y 402.273,Z 791.391,A -85,B 0,C 180,E1 -21935.106,E2 -21935.106} C_VEL
LIN {X 0,Y 406.787,Z 767.391,A -85,B 0,C 180,E1 -21935.751,E2 -21935.751} C_VEL
LIN {X 0,Y 409.842,Z 743.575,A -85,B 0,C 180,E1 -21936.222,E2 -21936.222} C_VEL
LIN {X 0,Y 415.159,Z 681.376,A -85,B 0,C 180,E1 -21937.228,E2 -21937.228} C_VEL
LIN {X 0,Y 415.386,Z 673.823,A -85,B 0,C 180,E1 -21937.476,E2 -21937.476} C_VEL
LIN {X 0,Y 414.627,Z 654.163,A -85,B 0,C 180,E1 -21938.583,E2 -21938.583} C_VEL
LIN {X 0,Y 414.9,Z 647.668,A -85,B 0,C 180,E1 -21938.782,E2 -21938.782} C_VEL
LIN {X 0,Y 422.541,Z 559.274,A -85,B 0,C 180,E1 -21940.185,E2 -21940.185} C_VEL
LIN {X 0,Y 416.843,Z 549.22,A -85,B 0,C 180,E1 -21942.912,E2 -21942.912} C_VEL
LIN {X 0,Y 412.069,Z 541.213,A -85,B 0,C 180,E1 -21945.598,E2 -21945.598} C_VEL
LIN {X 0,Y 407.973,Z 534.388,A -85,B 0,C 180,E1 -21948.406,E2 -21948.406} C_VEL
LIN {X 0,Y 405.035,Z 529.771,A -85,B 0,C 180,E1 -21950.909,E2 -21950.909} C_VEL
LIN {X 0,Y 402.367,Z 525.305,A -85,B 0,C 180,E1 -21954.009,E2 -21954.009} C_VEL
LIN {X 0,Y 400.08,Z 520.669,A -85,B 0,C 180,E1 -21960.859,E2 -21960.859} C_VEL
LIN {X 0,Y 402.66,Z 525.801,A -85,B 0,C 180,E1 -21968.065,E2 -21968.065} C_VEL
LIN {X 0,Y 405.249,Z 530.019,A -85,B 0,C 180,E1 -21970.952,E2 -21970.952} C_VEL
LIN {X 0,Y 408.874,Z 535.96,A -85,B 0,C 180,E1 -21973.938,E2 -21973.938} C_VEL
LIN {X 0,Y 412.058,Z 541.171,A -85,B 0,C 180,E1 -21976.059,E2 -21976.059} C_VEL
LIN {X 0,Y 414.568,Z 545.618,A -85,B 0,C 180,E1 -21977.547,E2 -21977.547} C_VEL
LIN {X 0,Y 419.938,Z 556.451,A -85,B 0,C 180,E1 -21980.379,E2 -21980.379} C_VEL
LIN {X 0,Y 422.458,Z 562.256,A -85,B 0,C 180,E1 -21981.591,E2 -21981.591} C_VEL
LIN {X 0,Y 405.55,Z 756.488,A -85,B 0,C 180,E1 -21984.679,E2 -21984.679} C_VEL
LIN {X 0,Y 401.596,Z 783.183,A -85,B 0,C 180,E1 -21985.224,E2 -21985.224} C_VEL
LIN {X 0,Y 397.168,Z 804.654,A -85,B 0,C 180,E1 -21985.787,E2 -21985.787} C_VEL
LIN {X 0,Y 390.88,Z 829.007,A -85,B 0,C 180,E1 -21986.615,E2 -21986.615} C_VEL
LIN {X 0,Y 384.797,Z 848.536,A -85,B 0,C 180,E1 -21987.454,E2 -21987.454} C_VEL
LIN {X 0,Y 376.997,Z 870.507,A -85,B 0,C 180,E1 -21988.611,E2 -21988.611} C_VEL
LIN {X 0,Y 367.944,Z 892.434,A -85,B 0,C 180,E1 -21990.057,E2 -21990.057} C_VEL
LIN {X 0,Y 359.151,Z 911.567,A -85,B 0,C 180,E1 -21991.579,E2 -21991.579} C_VEL
LIN {X 0,Y 348.624,Z 932.171,A -85,B 0,C 180,E1 -21993.588,E2 -21993.588} C_VEL
LIN {X 0,Y 339.031,Z 949.387,A -85,B 0,C 180,E1 -21995.616,E2 -21995.616} C_VEL
LIN {X 0,Y 327.607,Z 968.363,A -85,B 0,C 180,E1 -21998.336,E2 -21998.336} C_VEL
LIN {X 0,Y 317.878,Z 983.509,A -85,B 0,C 180,E1 -22000.981,E2 -22000.981} C_VEL
LIN {X 0,Y 306.832,Z 999.938,A -85,B 0,C 180,E1 -22004.478,E2 -22004.478} C_VEL
LIN {X 0,Y 297.875,Z 1012.757,A -85,B 0,C 180,E1 -22007.829,E2 -22007.829} C_VEL
LIN {X 0,Y 288.76,Z 1025.735,A -85,B 0,C 180,E1 -22011.949,E2 -22011.949} C_VEL
LIN {X 0,Y 281.408,Z 1036.225,A -85,B 0,C 180,E1 -22016.093,E2 -22016.093} C_VEL
LIN {X 0,Y 274.916,Z 1046.06,A -85,B 0,C 180,E1 -22020.832,E2 -22020.832} C_VEL
LIN {X 0,Y 270.052,Z 1053.953,A -85,B 0,C 180,E1 -22025.733,E2 -22025.733} C_VEL
LIN {X 0,Y 266.872,Z 1060.095,A -85,B 0,C 180,E1 -22030.521,E2 -22030.521} C_VEL
LIN {X 0,Y 264.805,Z 1065.257,A -85,B 0,C 180,E1 -22036.015,E2 -22036.015} C_VEL
LIN {X 0,Y 264.108,Z 1068.114,A -85,B 0,C 180,E1 -22040.411,E2 -22040.411} C_VEL
LIN {X 0,Y 263.971,Z 1069.877,A -85,B 0,C 180,E1 -22044.784,E2 -22044.784} C_VEL
LIN {X 0,Y 264.002,Z 1070.551,A -85,B 0,C 180,E1 -22049.349,E2 -22049.349} C_VEL
LIN {X 0,Y 263.978,Z 1069.85,A -85,B 0,C 180,E1 -22053.909,E2 -22053.909} C_VEL
LIN {X 0,Y 264.016,Z 1068.183,A -85,B 0,C 180,E1 -22058.055,E2 -22058.055} C_VEL
LIN {X 0,Y 264.469,Z 1065.337,A -85,B 0,C 180,E1 -22062.445,E2 -22062.445} C_VEL
LIN {X 0,Y 265.983,Z 1060.421,A -85,B 0,C 180,E1 -22067.728,E2 -22067.728} C_VEL
LIN {X 0,Y 268.609,Z 1054.286,A -85,B 0,C 180,E1 -22072.545,E2 -22072.545} C_VEL
LIN {X 0,Y 272.852,Z 1046.342,A -85,B 0,C 180,E1 -22077.522,E2 -22077.522} C_VEL
LIN {X 0,Y 278.653,Z 1036.514,A -85,B 0,C 180,E1 -22082.32,E2 -22082.32} C_VEL
LIN {X 0,Y 285.398,Z 1025.951,A -85,B 0,C 180,E1 -22086.555,E2 -22086.555} C_VEL
LIN {X 0,Y 293.875,Z 1012.853,A -85,B 0,C 180,E1 -22090.788,E2 -22090.788} C_VEL
LIN {X 0,Y 302.339,Z 999.862,A -85,B 0,C 180,E1 -22094.252,E2 -22094.252} C_VEL
LIN {X 0,Y 312.68,Z 983.49,A -85,B 0,C 180,E1 -22097.814,E2 -22097.814} C_VEL
LIN {X 0,Y 321.585,Z 968.835,A -85,B 0,C 180,E1 -22100.452,E2 -22100.452} C_VEL
LIN {X 0,Y 332.759,Z 949.297,A -85,B 0,C 180,E1 -22103.35,E2 -22103.35} C_VEL
LIN {X 0,Y 341.818,Z 932.27,A -85,B 0,C 180,E1 -22105.424,E2 -22105.424} C_VEL
LIN {X 0,Y 352.329,Z 910.696,A -85,B 0,C 180,E1 -22107.596,E2 -22107.596} C_VEL
LIN {X 0,Y 360.6,Z 891.945,A -85,B 0,C 180,E1 -22109.137,E2 -22109.137} C_VEL
LIN {X 0,Y 369.484,Z 869.422,A -85,B 0,C 180,E1 -22110.671,E2 -22110.671} C_VEL
LIN {X 0,Y 376.626,Z 848.549,A -85,B 0,C 180,E1 -22111.813,E2 -22111.813} C_VEL
LIN {X 0,Y 383.323,Z 826.187,A -85,B 0,C 180,E1 -22112.809,E2 -22112.809} C_VEL
LIN {X 0,Y 388.947,Z 802.957,A -85,B 0,C 180,E1 -22113.609,E2 -22113.609} C_VEL
LIN {X 0,Y 393.386,Z 780.337,A -85,B 0,C 180,E1 -22114.217,E2 -22114.217} C_VEL
LIN {X 0,Y 396.831,Z 754.948,A -85,B 0,C 180,E1 -22114.739,E2 -22114.739} C_VEL
LIN {X 0,Y 413.463,Z 555.447,A -85,B 0,C 180,E1 -22117.985,E2 -22117.985} C_VEL
LIN {X 0,Y 407.879,Z 543.86,A -85,B 0,C 180,E1 -22120.45,E2 -22120.45} C_VEL
LIN {X 0,Y 403.629,Z 535.552,A -85,B 0,C 180,E1 -22122.557,E2 -22122.557} C_VEL
LIN {X 0,Y 399.117,Z 528.224,A -85,B 0,C 180,E1 -22125.046,E2 -22125.046} C_VEL
LIN {X 0,Y 395.939,Z 523.174,A -85,B 0,C 180,E1 -22127.086,E2 -22127.086} C_VEL
LIN {X 0,Y 394.08,Z 520.288,A -85,B 0,C 180,E1 -22128.437,E2 -22128.437} C_VEL
LIN {X 0,Y 391.375,Z 516.041,A -85,B 0,C 180,E1 -22130.738,E2 -22130.738} C_VEL
LIN {X 0,Y 388.773,Z 511.721,A -85,B 0,C 180,E1 -22133.651,E2 -22133.651} C_VEL
LIN {X 0,Y 386.056,Z 506.398,A -85,B 0,C 180,E1 -22141.336,E2 -22141.336} C_VEL
LIN {X 0,Y 388.849,Z 511.898,A -85,B 0,C 180,E1 -22148.875,E2 -22148.875} C_VEL
LIN {X 0,Y 391.663,Z 516.343,A -85,B 0,C 180,E1 -22151.934,E2 -22151.934} C_VEL
LIN {X 0,Y 395.503,Z 522.476,A -85,B 0,C 180,E1 -22155.026,E2 -22155.026} C_VEL
LIN {X 0,Y 399.083,Z 528.109,A -85,B 0,C 180,E1 -22157.347,E2 -22157.347} C_VEL
LIN {X 0,Y 403.868,Z 535.881,A -85,B 0,C 180,E1 -22159.978,E2 -22159.978} C_VEL
LIN {X 0,Y 409.546,Z 545.579,A -85,B 0,C 180,E1 -22162.656,E2 -22162.656} C_VEL
LIN {X 0,Y 413.588,Z 552.964,A -85,B 0,C 180,E1 -22164.365,E2 -22164.365} C_VEL
LIN {X 0,Y 397.244,Z 747.418,A -85,B 0,C 180,E1 -22167.512,E2 -22167.512} C_VEL
LIN {X 0,Y 393.508,Z 773.872,A -85,B 0,C 180,E1 -22168.092,E2 -22168.092} C_VEL
LIN {X 0,Y 389.503,Z 794.561,A -85,B 0,C 180,E1 -22168.697,E2 -22168.697} C_VEL
LIN {X 0,Y 383.572,Z 819.078,A -85,B 0,C 180,E1 -22169.615,E2 -22169.615} C_VEL
LIN {X 0,Y 377.502,Z 839.643,A -85,B 0,C 180,E1 -22170.59,E2 -22170.59} C_VEL
LIN {X 0,Y 370.179,Z 861.348,A -85,B 0,C 180,E1 -22171.843,E2 -22171.843} C_VEL
LIN {X 0,Y 361.567,Z 883.06,A -85,B 0,C 180,E1 -22173.389,E2 -22173.389} C_VEL
LIN {X 0,Y 352.648,Z 903.392,A -85,B 0,C 180,E1 -22175.141,E2 -22175.141} C_VEL
LIN {X 0,Y 342.827,Z 923.22,A -85,B 0,C 180,E1 -22177.228,E2 -22177.228} C_VEL
LIN {X 0,Y 333.395,Z 940.87,A -85,B 0,C 180,E1 -22179.455,E2 -22179.455} C_VEL
LIN {X 0,Y 322.96,Z 958.778,A -85,B 0,C 180,E1 -22182.209,E2 -22182.209} C_VEL
LIN {X 0,Y 313.764,Z 973.718,A -85,B 0,C 180,E1 -22184.971,E2 -22184.971} C_VEL
LIN {X 0,Y 303.526,Z 989.517,A -85,B 0,C 180,E1 -22188.537,E2 -22188.537} C_VEL
LIN {X 0,Y 295.212,Z 1001.951,A -85,B 0,C 180,E1 -22191.944,E2 -22191.944} C_VEL
LIN {X 0,Y 286.477,Z 1014.88,A -85,B 0,C 180,E1 -22196.292,E2 -22196.292} C_VEL
LIN {X 0,Y 280.076,Z 1024.445,A -85,B 0,C 180,E1 -22200.249,E2 -22200.249} C_VEL
LIN {X 0,Y 273.93,Z 1034.106,A -85,B 0,C 180,E1 -22205.18,E2 -22205.18} C_VEL
LIN {X 0,Y 269.738,Z 1041.252,A -85,B 0,C 180,E1 -22209.834,E2 -22209.834} C_VEL
LIN {X 0,Y 266.65,Z 1047.491,A -85,B 0,C 180,E1 -22215.005,E2 -22215.005} C_VEL
LIN {X 0,Y 264.949,Z 1051.769,A -85,B 0,C 180,E1 -22220.003,E2 -22220.003} C_VEL
LIN {X 0,Y 264.265,Z 1054.38,A -85,B 0,C 180,E1 -22224.354,E2 -22224.354} C_VEL
LIN {X 0,Y 264.029,Z 1056.114,A -85,B 0,C 180,E1 -22229.349,E2 -22229.349} C_VEL
LIN {X 0,Y 264.015,Z 1056.357,A -85,B 0,C 180,E1 -22233.909,E2 -22233.909} C_VEL
LIN {X 0,Y 264.155,Z 1055.619,A -85,B 0,C 180,E1 -22238.051,E2 -22238.051} C_VEL
LIN {X 0,Y 264.623,Z 1053.931,A -85,B 0,C 180,E1 -22242.216,E2 -22242.216} C_VEL
LIN {X 0,Y 266.023,Z 1050.613,A -85,B 0,C 180,E1 -22247.311,E2 -22247.311} C_VEL
LIN {X 0,Y 268.588,Z 1045.68,A -85,B 0,C 180,E1 -22252.316,E2 -22252.316} C_VEL
LIN {X 0,Y 272.399,Z 1039.575,A -85,B 0,C 180,E1 -22257.076,E2 -22257.076} C_VEL
LIN {X 0,Y 278.174,Z 1031.101,A -85,B 0,C 180,E1 -22262.14,E2 -22262.14} C_VEL
LIN {X 0,Y 284.319,Z 1022.565,A -85,B 0,C 180,E1 -22266.215,E2 -22266.215} C_VEL
LIN {X 0,Y 293.288,Z 1010.366,A -85,B 0,C 180,E1 -22270.887,E2 -22270.887} C_VEL
LIN {X 0,Y 301.557,Z 999.016,A -85,B 0,C 180,E1 -22274.397,E2 -22274.397} C_VEL
LIN {X 0,Y 311.843,Z 984.569,A -85,B 0,C 180,E1 -22278.063,E2 -22278.063} C_VEL
LIN {X 0,Y 321.55,Z 970.226,A -85,B 0,C 180,E1 -22281.023,E2 -22281.023} C_VEL
LIN {X 0,Y 332.159,Z 953.804,A -85,B 0,C 180,E1 -22283.842,E2 -22283.842} C_VEL
LIN {X 0,Y 342.234,Z 936.819,A -85,B 0,C 180,E1 -22286.223,E2 -22286.223} C_VEL
LIN {X 0,Y 352.025,Z 919.162,A -85,B 0,C 180,E1 -22288.3,E2 -22288.3} C_VEL
LIN {X 0,Y 361.813,Z 899.568,A -85,B 0,C 180,E1 -22290.199,E2 -22290.199} C_VEL
LIN {X 0,Y 369.855,Z 881.819,A -85,B 0,C 180,E1 -22291.64,E2 -22291.64} C_VEL
LIN {X 0,Y 378.855,Z 859.592,A -85,B 0,C 180,E1 -22293.134,E2 -22293.134} C_VEL
LIN {X 0,Y 385.95,Z 839.194,A -85,B 0,C 180,E1 -22294.257,E2 -22294.257} C_VEL
LIN {X 0,Y 392.93,Z 816.1,A -85,B 0,C 180,E1 -22295.293,E2 -22295.293} C_VEL
LIN {X 0,Y 398.61,Z 792.605,A -85,B 0,C 180,E1 -22296.11,E2 -22296.11} C_VEL
LIN {X 0,Y 403.197,Z 769.107,A -85,B 0,C 180,E1 -22296.745,E2 -22296.745} C_VEL
LIN {X 0,Y 406.468,Z 744.491,A -85,B 0,C 180,E1 -22297.234,E2 -22297.234} C_VEL
LIN {X 0,Y 414.9,Z 647.668,A -85,B 0,C 180,E1 -22298.782,E2 -22298.782} C_VEL
LIN {X 0,Y 415.177,Z 640.115,A -85,B 0,C 180,E1 -22299.03,E2 -22299.03} C_VEL
LIN {X 0,Y 414.624,Z 620.462,A -85,B 0,C 180,E1 -22300.143,E2 -22300.143} C_VEL
LIN {X 0,Y 414.936,Z 613.967,A -85,B 0,C 180,E1 -22300.341,E2 -22300.341} C_VEL
LIN {X 0,Y 419.36,Z 564.343,A -85,B 0,C 180,E1 -22301.115,E2 -22301.115} C_VEL
LIN {X 0,Y 413.72,Z 554.136,A -85,B 0,C 180,E1 -22304.007,E2 -22304.007} C_VEL
LIN {X 0,Y 408.97,Z 546.064,A -85,B 0,C 180,E1 -22306.929,E2 -22306.929} C_VEL
LIN {X 0,Y 405.997,Z 541.23,A -85,B 0,C 180,E1 -22309.14,E2 -22309.14} C_VEL
LIN {X 0,Y 403.759,Z 537.481,A -85,B 0,C 180,E1 -22311.168,E2 -22311.168} C_VEL
LIN {X 0,Y 401.18,Z 533.109,A -85,B 0,C 180,E1 -22314.278,E2 -22314.278} C_VEL
LIN {X 0,Y 399.103,Z 528.618,A -85,B 0,C 180,E1 -22320.861,E2 -22320.861} C_VEL
LIN {X 0,Y 401.522,Z 533.618,A -85,B 0,C 180,E1 -22327.872,E2 -22327.872} C_VEL
LIN {X 0,Y 404.548,Z 538.8,A -85,B 0,C 180,E1 -22331.26,E2 -22331.26} C_VEL
LIN {X 0,Y 407.596,Z 543.839,A -85,B 0,C 180,E1 -22333.766,E2 -22333.766} C_VEL
LIN {X 0,Y 410.841,Z 549.26,A -85,B 0,C 180,E1 -22335.963,E2 -22335.963} C_VEL
LIN {X 0,Y 413.597,Z 554.533,A -85,B 0,C 180,E1 -22337.626,E2 -22337.626} C_VEL
LIN {X 0,Y 418.407,Z 564.676,A -85,B 0,C 180,E1 -22340.201,E2 -22340.201} C_VEL
LIN {X 0,Y 419.27,Z 566.769,A -85,B 0,C 180,E1 -22340.637,E2 -22340.637} C_VEL
LIN {X 0,Y 402.379,Z 756.349,A -85,B 0,C 180,E1 -22343.633,E2 -22343.633} C_VEL
LIN {X 0,Y 398.355,Z 783.014,A -85,B 0,C 180,E1 -22344.171,E2 -22344.171} C_VEL
LIN {X 0,Y 393.875,Z 804.37,A -85,B 0,C 180,E1 -22344.723,E2 -22344.723} C_VEL
LIN {X 0,Y 387.35,Z 829.141,A -85,B 0,C 180,E1 -22345.553,E2 -22345.553} C_VEL
LIN {X 0,Y 380.773,Z 849.756,A -85,B 0,C 180,E1 -22346.434,E2 -22346.434} C_VEL
LIN {X 0,Y 372.452,Z 872.443,A -85,B 0,C 180,E1 -22347.635,E2 -22347.635} C_VEL
LIN {X 0,Y 363.591,Z 893.249,A -85,B 0,C 180,E1 -22349.013,E2 -22349.013} C_VEL
LIN {X 0,Y 353.746,Z 914.085,A -85,B 0,C 180,E1 -22350.68,E2 -22350.68} C_VEL
LIN {X 0,Y 343.195,Z 933.886,A -85,B 0,C 180,E1 -22352.649,E2 -22352.649} C_VEL
LIN {X 0,Y 332.307,Z 952.812,A -85,B 0,C 180,E1 -22354.922,E2 -22354.922} C_VEL
LIN {X 0,Y 321.361,Z 970.13,A -85,B 0,C 180,E1 -22357.494,E2 -22357.494} C_VEL
LIN {X 0,Y 310.847,Z 985.952,A -85,B 0,C 180,E1 -22360.328,E2 -22360.328} C_VEL
LIN {X 0,Y 300.095,Z 1001.191,A -85,B 0,C 180,E1 -22363.695,E2 -22363.695} C_VEL
LIN {X 0,Y 290.873,Z 1013.903,A -85,B 0,C 180,E1 -22367.107,E2 -22367.107} C_VEL
LIN {X 0,Y 281.093,Z 1027.145,A -85,B 0,C 180,E1 -22371.501,E2 -22371.501} C_VEL
LIN {X 0,Y 273.756,Z 1037.209,A -85,B 0,C 180,E1 -22375.636,E2 -22375.636} C_VEL
LIN {X 0,Y 266.454,Z 1047.686,A -85,B 0,C 180,E1 -22381.048,E2 -22381.048} C_VEL
LIN {X 0,Y 262.003,Z 1054.7,A -85,B 0,C 180,E1 -22385.659,E2 -22385.659} C_VEL
LIN {X 0,Y 258.361,Z 1061.504,A -85,B 0,C 180,E1 -22391.475,E2 -22391.475} C_VEL
LIN {X 0,Y 256.739,Z 1065.554,A -85,B 0,C 180,E1 -22396.257,E2 -22396.257} C_VEL
LIN {X 0,Y 256.063,Z 1068.423,A -85,B 0,C 180,E1 -22401.09,E2 -22401.09} C_VEL
LIN {X 0,Y 255.972,Z 1069.995,A -85,B 0,C 180,E1 -22405.968,E2 -22405.968} C_VEL
LIN {X 0,Y 256.011,Z 1070.223,A -85,B 0,C 180,E1 -22410.448,E2 -22410.448} C_VEL
LIN {X 0,Y 255.978,Z 1069.488,A -85,B 0,C 180,E1 -22414.481,E2 -22414.481} C_VEL
LIN {X 0,Y 256.043,Z 1067.836,A -85,B 0,C 180,E1 -22418.534,E2 -22418.534} C_VEL
LIN {X 0,Y 256.577,Z 1064.934,A -85,B 0,C 180,E1 -22423.063,E2 -22423.063} C_VEL
LIN {X 0,Y 258.386,Z 1059.646,A -85,B 0,C 180,E1 -22428.735,E2 -22428.735} C_VEL
LIN {X 0,Y 261.178,Z 1053.714,A -85,B 0,C 180,E1 -22433.463,E2 -22433.463} C_VEL
LIN {X 0,Y 265.753,Z 1045.722,A -85,B 0,C 180,E1 -22438.544,E2 -22438.544} C_VEL
LIN {X 0,Y 271.893,Z 1035.899,A -85,B 0,C 180,E1 -22443.405,E2 -22443.405} C_VEL
LIN {X 0,Y 279.514,Z 1024.592,A -85,B 0,C 180,E1 -22447.973,E2 -22447.973} C_VEL
LIN {X 0,Y 288.077,Z 1011.898,A -85,B 0,C 180,E1 -22452.058,E2 -22452.058} C_VEL
LIN {X 0,Y 297.444,Z 998.121,A -85,B 0,C 180,E1 -22455.727,E2 -22455.727} C_VEL
LIN {X 0,Y 307.334,Z 982.906,A -85,B 0,C 180,E1 -22459.007,E2 -22459.007} C_VEL
LIN {X 0,Y 317.323,Z 966.988,A -85,B 0,C 180,E1 -22461.859,E2 -22461.859} C_VEL
LIN {X 0,Y 328.221,Z 948.363,A -85,B 0,C 180,E1 -22464.578,E2 -22464.578} C_VEL
LIN {X 0,Y 337.928,Z 930.566,A -85,B 0,C 180,E1 -22466.722,E2 -22466.722} C_VEL
LIN {X 0,Y 348.354,Z 909.534,A -85,B 0,C 180,E1 -22468.799,E2 -22468.799} C_VEL
LIN {X 0,Y 356.783,Z 890.808,A -85,B 0,C 180,E1 -22470.317,E2 -22470.317} C_VEL
LIN {X 0,Y 366.174,Z 867.228,A -85,B 0,C 180,E1 -22471.884,E2 -22471.884} C_VEL
LIN {X 0,Y 373.231,Z 846.885,A -85,B 0,C 180,E1 -22472.97,E2 -22472.97} C_VEL
LIN {X 0,Y 380.238,Z 823.446,A -85,B 0,C 180,E1 -22473.976,E2 -22473.976} C_VEL
LIN {X 0,Y 385.56,Z 801.659,A -85,B 0,C 180,E1 -22474.703,E2 -22474.703} C_VEL
LIN {X 0,Y 390.306,Z 777.572,A -85,B 0,C 180,E1 -22475.331,E2 -22475.331} C_VEL
LIN {X 0,Y 393.539,Z 752.897,A -85,B 0,C 180,E1 -22475.82,E2 -22475.82} C_VEL
LIN {X 0,Y 410.004,Z 559.968,A -85,B 0,C 180,E1 -22478.936,E2 -22478.936} C_VEL
LIN {X 0,Y 405.405,Z 550.158,A -85,B 0,C 180,E1 -22481.075,E2 -22481.075} C_VEL
LIN {X 0,Y 401.623,Z 542.572,A -85,B 0,C 180,E1 -22483.028,E2 -22483.028} C_VEL
LIN {X 0,Y 397.306,Z 535.4,A -85,B 0,C 180,E1 -22485.498,E2 -22485.498} C_VEL
LIN {X 0,Y 393.39,Z 528.806,A -85,B 0,C 180,E1 -22488.193,E2 -22488.193} C_VEL
LIN {X 0,Y 390.082,Z 523.752,A -85,B 0,C 180,E1 -22491.004,E2 -22491.004} C_VEL
LIN {X 0,Y 387.344,Z 519.272,A -85,B 0,C 180,E1 -22494.222,E2 -22494.222} C_VEL
LIN {X 0,Y 385.078,Z 514.364,A -85,B 0,C 180,E1 -22501.339,E2 -22501.339} C_VEL
LIN {X 0,Y 387.752,Z 519.847,A -85,B 0,C 180,E1 -22508.751,E2 -22508.751} C_VEL
LIN {X 0,Y 390.984,Z 525.13,A -85,B 0,C 180,E1 -22512.255,E2 -22512.255} C_VEL
LIN {X 0,Y 394.105,Z 530.18,A -85,B 0,C 180,E1 -22514.773,E2 -22514.773} C_VEL
LIN {X 0,Y 397.509,Z 535.663,A -85,B 0,C 180,E1 -22517.04,E2 -22517.04} C_VEL
LIN {X 0,Y 402.393,Z 543.816,A -85,B 0,C 180,E1 -22519.789,E2 -22519.789} C_VEL
LIN {X 0,Y 407.755,Z 553.293,A -85,B 0,C 180,E1 -22522.377,E2 -22522.377} C_VEL
LIN {X 0,Y 410.091,Z 557.754,A -85,B 0,C 180,E1 -22523.411,E2 -22523.411} C_VEL
LIN {X 0,Y 393.75,Z 747.589,A -85,B 0,C 180,E1 -22526.469,E2 -22526.469} C_VEL
LIN {X 0,Y 389.94,Z 774.061,A -85,B 0,C 180,E1 -22527.043,E2 -22527.043} C_VEL
LIN {X 0,Y 385.842,Z 794.82,A -85,B 0,C 180,E1 -22527.643,E2 -22527.643} C_VEL
LIN {X 0,Y 380.057,Z 818.404,A -85,B 0,C 180,E1 -22528.512,E2 -22528.512} C_VEL
LIN {X 0,Y 373.496,Z 840.196,A -85,B 0,C 180,E1 -22529.534,E2 -22529.534} C_VEL
LIN {X 0,Y 365.661,Z 862.774,A -85,B 0,C 180,E1 -22530.838,E2 -22530.838} C_VEL
LIN {X 0,Y 357.137,Z 883.691,A -85,B 0,C 180,E1 -22532.327,E2 -22532.327} C_VEL
LIN {X 0,Y 347.807,Z 904.404,A -85,B 0,C 180,E1 -22534.111,E2 -22534.111} C_VEL
LIN {X 0,Y 338.006,Z 923.619,A -85,B 0,C 180,E1 -22536.139,E2 -22536.139} C_VEL
LIN {X 0,Y 328.041,Z 941.749,A -85,B 0,C 180,E1 -22538.432,E2 -22538.432} C_VEL
LIN {X 0,Y 317.428,Z 959.357,A -85,B 0,C 180,E1 -22541.163,E2 -22541.163} C_VEL
LIN {X 0,Y 308.072,Z 974.064,A -85,B 0,C 180,E1 -22543.902,E2 -22543.902} C_VEL
LIN {X 0,Y 297.471,Z 989.842,A -85,B 0,C 180,E1 -22547.498,E2 -22547.498} C_VEL
LIN {X 0,Y 288.838,Z 1002.266,A -85,B 0,C 180,E1 -22550.947,E2 -22550.947} C_VEL
LIN {X 0,Y 279.726,Z 1015.178,A -85,B 0,C 180,E1 -22555.365,E2 -22555.365} C_VEL
LIN {X 0,Y 273.027,Z 1024.734,A -85,B 0,C 180,E1 -22559.399,E2 -22559.399} C_VEL
LIN {X 0,Y 266.562,Z 1034.378,A -85,B 0,C 180,E1 -22564.445,E2 -22564.445} C_VEL
LIN {X 0,Y 262.128,Z 1041.515,A -85,B 0,C 180,E1 -22569.222,E2 -22569.222} C_VEL
LIN {X 0,Y 258.842,Z 1047.739,A -85,B 0,C 180,E1 -22574.541,E2 -22574.541} C_VEL
LIN {X 0,Y 257.024,Z 1052.009,A -85,B 0,C 180,E1 -22579.691,E2 -22579.691} C_VEL
LIN {X 0,Y 256.283,Z 1054.626,A -85,B 0,C 180,E1 -22584.206,E2 -22584.206} C_VEL
LIN {X 0,Y 256.033,Z 1056.331,A -85,B 0,C 180,E1 -22589.329,E2 -22589.329} C_VEL
LIN {X 0,Y 256.02,Z 1056.568,A -85,B 0,C 180,E1 -22594.031,E2 -22594.031} C_VEL
LIN {X 0,Y 256.16,Z 1055.889,A -85,B 0,C 180,E1 -22598.078,E2 -22598.078} C_VEL
LIN {X 0,Y 256.653,Z 1054.24,A -85,B 0,C 180,E1 -22602.373,E2 -22602.373} C_VEL
LIN {X 0,Y 258.148,Z 1050.947,A -85,B 0,C 180,E1 -22607.666,E2 -22607.666} C_VEL
LIN {X 0,Y 260.988,Z 1045.859,A -85,B 0,C 180,E1 -22613.003,E2 -22613.003} C_VEL
LIN {X 0,Y 265.062,Z 1039.748,A -85,B 0,C 180,E1 -22617.889,E2 -22617.889} C_VEL
LIN {X 0,Y 271.19,Z 1031.258,A -85,B 0,C 180,E1 -22623.071,E2 -22623.071} C_VEL
LIN {X 0,Y 277.802,Z 1022.544,A -85,B 0,C 180,E1 -22627.302,E2 -22627.302} C_VEL
LIN {X 0,Y 287.066,Z 1010.498,A -85,B 0,C 180,E1 -22631.972,E2 -22631.972} C_VEL
LIN {X 0,Y 295.691,Z 999.138,A -85,B 0,C 180,E1 -22635.521,E2 -22635.521} C_VEL
LIN {X 0,Y 306.633,Z 984.305,A -85,B 0,C 180,E1 -22639.294,E2 -22639.294} C_VEL
LIN {X 0,Y 316.473,Z 970.246,A -85,B 0,C 180,E1 -22642.197,E2 -22642.197} C_VEL
LIN {X 0,Y 327.547,Z 953.575,A -85,B 0,C 180,E1 -22645.049,E2 -22645.049} C_VEL
LIN {X 0,Y 337.882,Z 936.625,A -85,B 0,C 180,E1 -22647.412,E2 -22647.412} C_VEL
LIN {X 0,Y 348.112,Z 918.633,A -85,B 0,C 180,E1 -22649.508,E2 -22649.508} C_VEL
LIN {X 0,Y 358.177,Z 898.826,A -85,B 0,C 180,E1 -22651.397,E2 -22651.397} C_VEL
LIN {X 0,Y 366.425,Z 880.976,A -85,B 0,C 180,E1 -22652.82,E2 -22652.82} C_VEL
LIN {X 0,Y 376,Z 857.489,A -85,B 0,C 180,E1 -22654.355,E2 -22654.355} C_VEL
LIN {X 0,Y 382.742,Z 838.351,A -85,B 0,C 180,E1 -22655.385,E2 -22655.385} C_VEL
LIN {X 0,Y 389.93,Z 814.649,A -85,B 0,C 180,E1 -22656.42,E2 -22656.42} C_VEL
LIN {X 0,Y 395.432,Z 792.19,A -85,B 0,C 180,E1 -22657.184,E2 -22657.184} C_VEL
LIN {X 0,Y 400.132,Z 768.278,A -85,B 0,C 180,E1 -22657.815,E2 -22657.815} C_VEL
LIN {X 0,Y 403.365,Z 744.104,A -85,B 0,C 180,E1 -22658.285,E2 -22658.285} C_VEL
LIN {X 0,Y 414.936,Z 613.967,A -85,B 0,C 180,E1 -22660.341,E2 -22660.341} C_VEL
LIN {X 0,Y 415.264,Z 606.416,A -85,B 0,C 180,E1 -22660.586,E2 -22660.586} C_VEL
LIN {X 0,Y 414.927,Z 586.769,A -85,B 0,C 180,E1 -22661.702,E2 -22661.702} C_VEL
LIN {X 0,Y 415.264,Z 580.278,A -85,B 0,C 180,E1 -22661.904,E2 -22661.904} C_VEL
LIN {X 0,Y 416.222,Z 569.318,A -85,B 0,C 180,E1 -22662.092,E2 -22662.092} C_VEL
LIN {X 0,Y 411.401,Z 560.533,A -85,B 0,C 180,E1 -22664.71,E2 -22664.71} C_VEL
LIN {X 0,Y 407.273,Z 553.31,A -85,B 0,C 180,E1 -22667.379,E2 -22667.379} C_VEL
LIN {X 0,Y 404.584,Z 548.791,A -85,B 0,C 180,E1 -22669.462,E2 -22669.462} C_VEL
LIN {X 0,Y 402.491,Z 545.19,A -85,B 0,C 180,E1 -22671.428,E2 -22671.428} C_VEL
LIN {X 0,Y 400.103,Z 540.993,A -85,B 0,C 180,E1 -22674.407,E2 -22674.407} C_VEL
LIN {X 0,Y 398.126,Z 536.577,A -85,B 0,C 180,E1 -22680.863,E2 -22680.863} C_VEL
LIN {X 0,Y 400.435,Z 541.558,A -85,B 0,C 180,E1 -22687.749,E2 -22687.749} C_VEL
LIN {X 0,Y 403.262,Z 546.497,A -85,B 0,C 180,E1 -22691.007,E2 -22691.007} C_VEL
LIN {X 0,Y 406.231,Z 551.55,A -85,B 0,C 180,E1 -22693.523,E2 -22693.523} C_VEL
LIN {X 0,Y 409.879,Z 557.729,A -85,B 0,C 180,E1 -22696.023,E2 -22696.023} C_VEL
LIN {X 0,Y 414.596,Z 567.79,A -85,B 0,C 180,E1 -22698.818,E2 -22698.818} C_VEL
LIN {X 0,Y 416.169,Z 571.629,A -85,B 0,C 180,E1 -22699.674,E2 -22699.674} C_VEL
LIN {X 0,Y 399.355,Z 756.105,A -85,B 0,C 180,E1 -22702.569,E2 -22702.569} C_VEL
LIN {X 0,Y 395.26,Z 782.795,A -85,B 0,C 180,E1 -22703.101,E2 -22703.101} C_VEL
LIN {X 0,Y 390.72,Z 804.085,A -85,B 0,C 180,E1 -22703.641,E2 -22703.641} C_VEL
LIN {X 0,Y 384.16,Z 828.617,A -85,B 0,C 180,E1 -22704.447,E2 -22704.447} C_VEL
LIN {X 0,Y 377.647,Z 848.72,A -85,B 0,C 180,E1 -22705.286,E2 -22705.286} C_VEL
LIN {X 0,Y 369.54,Z 870.622,A -85,B 0,C 180,E1 -22706.413,E2 -22706.413} C_VEL
LIN {X 0,Y 360.105,Z 892.442,A -85,B 0,C 180,E1 -22707.826,E2 -22707.826} C_VEL
LIN {X 0,Y 350.198,Z 913.003,A -85,B 0,C 180,E1 -22709.444,E2 -22709.444} C_VEL
LIN {X 0,Y 339.56,Z 932.615,A -85,B 0,C 180,E1 -22711.356,E2 -22711.356} C_VEL
LIN {X 0,Y 329.348,Z 949.968,A -85,B 0,C 180,E1 -22713.395,E2 -22713.395} C_VEL
LIN {X 0,Y 317.272,Z 968.784,A -85,B 0,C 180,E1 -22716.11,E2 -22716.11} C_VEL
LIN {X 0,Y 306.74,Z 984.149,A -85,B 0,C 180,E1 -22718.824,E2 -22718.824} C_VEL
LIN {X 0,Y 294.977,Z 1000.361,A -85,B 0,C 180,E1 -22722.357,E2 -22722.357} C_VEL
LIN {X 0,Y 285.344,Z 1013.128,A -85,B 0,C 180,E1 -22725.787,E2 -22725.787} C_VEL
LIN {X 0,Y 275.066,Z 1026.474,A -85,B 0,C 180,E1 -22730.225,E2 -22730.225} C_VEL
LIN {X 0,Y 267.462,Z 1036.371,A -85,B 0,C 180,E1 -22734.324,E2 -22734.324} C_VEL
LIN {X 0,Y 260.037,Z 1046.435,A -85,B 0,C 180,E1 -22739.498,E2 -22739.498} C_VEL
LIN {X 0,Y 254.873,Z 1053.939,A -85,B 0,C 180,E1 -22744.464,E2 -22744.464} C_VEL
LIN {X 0,Y 251.062,Z 1060.483,A -85,B 0,C 180,E1 -22749.97,E2 -22749.97} C_VEL
LIN {X 0,Y 248.95,Z 1065.028,A -85,B 0,C 180,E1 -22755.343,E2 -22755.343} C_VEL
LIN {X 0,Y 248.14,Z 1067.83,A -85,B 0,C 180,E1 -22760.022,E2 -22760.022} C_VEL
LIN {X 0,Y 247.973,Z 1069.677,A -85,B 0,C 180,E1 -22765.142,E2 -22765.142} C_VEL
LIN {X 0,Y 248.021,Z 1070.052,A -85,B 0,C 180,E1 -22770,E2 -22770} C_VEL
LIN {X 0,Y 247.98,Z 1069.335,A -85,B 0,C 180,E1 -22774.394,E2 -22774.394} C_VEL
LIN {X 0,Y 248.046,Z 1067.723,A -85,B 0,C 180,E1 -22778.578,E2 -22778.578} C_VEL
LIN {X 0,Y 248.608,Z 1064.852,A -85,B 0,C 180,E1 -22783.265,E2 -22783.265} C_VEL
LIN {X 0,Y 250.517,Z 1059.654,A -85,B 0,C 180,E1 -22789.104,E2 -22789.104} C_VEL
LIN {X 0,Y 253.457,Z 1053.765,A -85,B 0,C 180,E1 -22793.975,E2 -22793.975} C_VEL
LIN {X 0,Y 258.258,Z 1045.839,A -85,B 0,C 180,E1 -22799.198,E2 -22799.198} C_VEL
LIN {X 0,Y 264.773,Z 1035.947,A -85,B 0,C 180,E1 -22804.242,E2 -22804.242} C_VEL
LIN {X 0,Y 272.617,Z 1024.843,A -85,B 0,C 180,E1 -22808.843,E2 -22808.843} C_VEL
LIN {X 0,Y 281.51,Z 1012.236,A -85,B 0,C 180,E1 -22812.997,E2 -22812.997} C_VEL
LIN {X 0,Y 290.686,Z 999.228,A -85,B 0,C 180,E1 -22816.534,E2 -22816.534} C_VEL
LIN {X 0,Y 301.404,Z 983.427,A -85,B 0,C 180,E1 -22820.025,E2 -22820.025} C_VEL
LIN {X 0,Y 310.715,Z 969.08,A -85,B 0,C 180,E1 -22822.641,E2 -22822.641} C_VEL
LIN {X 0,Y 322.23,Z 950.24,A -85,B 0,C 180,E1 -22825.473,E2 -22825.473} C_VEL
LIN {X 0,Y 332.107,Z 932.701,A -85,B 0,C 180,E1 -22827.62,E2 -22827.62} C_VEL
LIN {X 0,Y 342.777,Z 912.085,A -85,B 0,C 180,E1 -22829.705,E2 -22829.705} C_VEL
LIN {X 0,Y 351.733,Z 892.799,A -85,B 0,C 180,E1 -22831.287,E2 -22831.287} C_VEL
LIN {X 0,Y 360.925,Z 870.794,A -85,B 0,C 180,E1 -22832.783,E2 -22832.783} C_VEL
LIN {X 0,Y 368.851,Z 848.64,A -85,B 0,C 180,E1 -22833.98,E2 -22833.98} C_VEL
LIN {X 0,Y 375.632,Z 826.938,A -85,B 0,C 180,E1 -22834.928,E2 -22834.928} C_VEL
LIN {X 0,Y 381.657,Z 803.273,A -85,B 0,C 180,E1 -22835.731,E2 -22835.731} C_VEL
LIN {X 0,Y 386.132,Z 781.442,A -85,B 0,C 180,E1 -22836.307,E2 -22836.307} C_VEL
LIN {X 0,Y 389.923,Z 755.233,A -85,B 0,C 180,E1 -22836.843,E2 -22836.843} C_VEL
LIN {X 0,Y 406.625,Z 564.396,A -85,B 0,C 180,E1 -22839.92,E2 -22839.92} C_VEL
LIN {X 0,Y 401.997,Z 554.312,A -85,B 0,C 180,E1 -22842.223,E2 -22842.223} C_VEL
LIN {X 0,Y 398.968,Z 548.318,A -85,B 0,C 180,E1 -22843.885,E2 -22843.885} C_VEL
LIN {X 0,Y 393.945,Z 539.834,A -85,B 0,C 180,E1 -22847.019,E2 -22847.019} C_VEL
LIN {X 0,Y 391.273,Z 535.532,A -85,B 0,C 180,E1 -22849.025,E2 -22849.025} C_VEL
LIN {X 0,Y 388.797,Z 531.461,A -85,B 0,C 180,E1 -22851.273,E2 -22851.273} C_VEL
LIN {X 0,Y 386.261,Z 527.154,A -85,B 0,C 180,E1 -22854.355,E2 -22854.355} C_VEL
LIN {X 0,Y 384.1,Z 522.33,A -85,B 0,C 180,E1 -22861.343,E2 -22861.343} C_VEL
LIN {X 0,Y 386.609,Z 527.665,A -85,B 0,C 180,E1 -22868.552,E2 -22868.552} C_VEL
LIN {X 0,Y 389.681,Z 532.832,A -85,B 0,C 180,E1 -22871.996,E2 -22871.996} C_VEL
LIN {X 0,Y 392.724,Z 537.899,A -85,B 0,C 180,E1 -22874.524,E2 -22874.524} C_VEL
LIN {X 0,Y 396.174,Z 543.574,A -85,B 0,C 180,E1 -22876.873,E2 -22876.873} C_VEL
LIN {X 0,Y 401.256,Z 552.273,A -85,B 0,C 180,E1 -22879.772,E2 -22879.772} C_VEL
LIN {X 0,Y 406.716,Z 562.494,A -85,B 0,C 180,E1 -22882.44,E2 -22882.44} C_VEL
LIN {X 0,Y 390.378,Z 747.862,A -85,B 0,C 180,E1 -22885.409,E2 -22885.409} C_VEL
LIN {X 0,Y 386.482,Z 774.375,A -85,B 0,C 180,E1 -22885.979,E2 -22885.979} C_VEL
LIN {X 0,Y 382.309,Z 795.094,A -85,B 0,C 180,E1 -22886.571,E2 -22886.571} C_VEL
LIN {X 0,Y 376.312,Z 819,A -85,B 0,C 180,E1 -22887.444,E2 -22887.444} C_VEL
LIN {X 0,Y 369.951,Z 839.739,A -85,B 0,C 180,E1 -22888.404,E2 -22888.404} C_VEL
LIN {X 0,Y 362.342,Z 861.385,A -85,B 0,C 180,E1 -22889.629,E2 -22889.629} C_VEL
LIN {X 0,Y 353.391,Z 883.053,A -85,B 0,C 180,E1 -22891.141,E2 -22891.141} C_VEL
LIN {X 0,Y 344.717,Z 901.951,A -85,B 0,C 180,E1 -22892.736,E2 -22892.736} C_VEL
LIN {X 0,Y 334.301,Z 922.216,A -85,B 0,C 180,E1 -22894.813,E2 -22894.813} C_VEL
LIN {X 0,Y 324.931,Z 938.89,A -85,B 0,C 180,E1 -22896.875,E2 -22896.875} C_VEL
LIN {X 0,Y 313.331,Z 957.889,A -85,B 0,C 180,E1 -22899.73,E2 -22899.73} C_VEL
LIN {X 0,Y 303.522,Z 972.849,A -85,B 0,C 180,E1 -22902.48,E2 -22902.48} C_VEL
LIN {X 0,Y 292.511,Z 988.789,A -85,B 0,C 180,E1 -22906.059,E2 -22906.059} C_VEL
LIN {X 0,Y 283.453,Z 1001.333,A -85,B 0,C 180,E1 -22909.529,E2 -22909.529} C_VEL
LIN {X 0,Y 274.208,Z 1013.96,A -85,B 0,C 180,E1 -22913.791,E2 -22913.791} C_VEL
LIN {X 0,Y 266.688,Z 1024.123,A -85,B 0,C 180,E1 -22918.086,E2 -22918.086} C_VEL
LIN {X 0,Y 259.994,Z 1033.612,A -85,B 0,C 180,E1 -22923.012,E2 -22923.012} C_VEL
LIN {X 0,Y 254.913,Z 1041.187,A -85,B 0,C 180,E1 -22928.122,E2 -22928.122} C_VEL
LIN {X 0,Y 251.523,Z 1047.053,A -85,B 0,C 180,E1 -22933.13,E2 -22933.13} C_VEL
LIN {X 0,Y 249.285,Z 1051.783,A -85,B 0,C 180,E1 -22938.665,E2 -22938.665} C_VEL
LIN {X 0,Y 248.38,Z 1054.512,A -85,B 0,C 180,E1 -22943.296,E2 -22943.296} C_VEL
LIN {X 0,Y 248.075,Z 1056.133,A -85,B 0,C 180,E1 -22947.69,E2 -22947.69} C_VEL
LIN {X 0,Y 248.004,Z 1056.84,A -85,B 0,C 180,E1 -22952.311,E2 -22952.311} C_VEL
LIN {X 0,Y 248.137,Z 1056.355,A -85,B 0,C 180,E1 -22957.409,E2 -22957.409} C_VEL
LIN {X 0,Y 248.642,Z 1054.659,A -85,B 0,C 180,E1 -22962.306,E2 -22962.306} C_VEL
LIN {X 0,Y 249.87,Z 1051.971,A -85,B 0,C 180,E1 -22966.985,E2 -22966.985} C_VEL
LIN {X 0,Y 252.833,Z 1046.979,A -85,B 0,C 180,E1 -22972.859,E2 -22972.859} C_VEL
LIN {X 0,Y 256.876,Z 1041.112,A -85,B 0,C 180,E1 -22977.846,E2 -22977.846} C_VEL
LIN {X 0,Y 263.072,Z 1033.015,A -85,B 0,C 180,E1 -22983.183,E2 -22983.183} C_VEL
LIN {X 0,Y 270.365,Z 1023.771,A -85,B 0,C 180,E1 -22987.873,E2 -22987.873} C_VEL
LIN {X 0,Y 279.2,Z 1012.904,A -85,B 0,C 180,E1 -22992.321,E2 -22992.321} C_VEL
LIN {X 0,Y 288.948,Z 1000.521,A -85,B 0,C 180,E1 -22996.322,E2 -22996.322} C_VEL
LIN {X 0,Y 299.389,Z 987.042,A -85,B 0,C 180,E1 -22999.89,E2 -22999.89} C_VEL
LIN {X 0,Y 310.24,Z 972.088,A -85,B 0,C 180,E1 -23003.063,E2 -23003.063} C_VEL
LIN {X 0,Y 320.673,Z 956.975,A -85,B 0,C 180,E1 -23005.72,E2 -23005.72} C_VEL
LIN {X 0,Y 332.382,Z 938.579,A -85,B 0,C 180,E1 -23008.357,E2 -23008.357} C_VEL
LIN {X 0,Y 341.93,Z 922.312,A -85,B 0,C 180,E1 -23010.285,E2 -23010.285} C_VEL
LIN {X 0,Y 353.262,Z 901.024,A -85,B 0,C 180,E1 -23012.366,E2 -23012.366} C_VEL
LIN {X 0,Y 362.036,Z 882.572,A -85,B 0,C 180,E1 -23013.845,E2 -23013.845} C_VEL
LIN {X 0,Y 371.461,Z 860.323,A -85,B 0,C 180,E1 -23015.314,E2 -23015.314} C_VEL
LIN {X 0,Y 379.053,Z 839.359,A -85,B 0,C 180,E1 -23016.442,E2 -23016.442} C_VEL
LIN {X 0,Y 386.254,Z 816.382,A -85,B 0,C 180,E1 -23017.445,E2 -23017.445} C_VEL
LIN {X 0,Y 392.125,Z 792.972,A -85,B 0,C 180,E1 -23018.238,E2 -23018.238} C_VEL
LIN {X 0,Y 396.905,Z 769.323,A -85,B 0,C 180,E1 -23018.858,E2 -23018.858} C_VEL
LIN {X 0,Y 400.292,Z 744.689,A -85,B 0,C 180,E1 -23019.335,E2 -23019.335} C_VEL
LIN {X 0,Y 415.264,Z 580.278,A -85,B 0,C 180,E1 -23021.904,E2 -23021.904} C_VEL
LIN {X 0,Y 415.202,Z 577.101,A -85,B 0,C 180,E1 -23022.096,E2 -23022.096} C_VEL
LIN {X 0,Y 414.493,Z 574.251,A -85,B 0,C 180,E1 -23022.539,E2 -23022.539} C_VEL
LIN {X 0,Y 412.986,Z 571.867,A -85,B 0,C 180,E1 -23023.316,E2 -23023.316} C_VEL
LIN {X 0,Y 410.26,Z 568.825,A -85,B 0,C 180,E1 -23024.749,E2 -23024.749} C_VEL
LIN {X 0,Y 405.888,Z 561,A -85,B 0,C 180,E1 -23027.624,E2 -23027.624} C_VEL
LIN {X 0,Y 403.184,Z 556.35,A -85,B 0,C 180,E1 -23029.786,E2 -23029.786} C_VEL
LIN {X 0,Y 401.232,Z 552.898,A -85,B 0,C 180,E1 -23031.689,E2 -23031.689} C_VEL
LIN {X 0,Y 399.029,Z 548.877,A -85,B 0,C 180,E1 -23034.536,E2 -23034.536} C_VEL
LIN {X 0,Y 397.148,Z 544.545,A -85,B 0,C 180,E1 -23040.866,E2 -23040.866} C_VEL
LIN {X 0,Y 399.305,Z 549.372,A -85,B 0,C 180,E1 -23047.554,E2 -23047.554} C_VEL
LIN {X 0,Y 402.053,Z 554.34,A -85,B 0,C 180,E1 -23050.822,E2 -23050.822} C_VEL
LIN {X 0,Y 404.963,Z 559.417,A -85,B 0,C 180,E1 -23053.348,E2 -23053.348} C_VEL
LIN {X 0,Y 408.355,Z 565.354,A -85,B 0,C 180,E1 -23055.735,E2 -23055.735} C_VEL
LIN {X 0,Y 413.221,Z 576.035,A -85,B 0,C 180,E1 -23058.686,E2 -23058.686} C_VEL
LIN {X 0,Y 396.472,Z 755.864,A -85,B 0,C 180,E1 -23061.489,E2 -23061.489} C_VEL
LIN {X 0,Y 392.307,Z 782.562,A -85,B 0,C 180,E1 -23062.013,E2 -23062.013} C_VEL
LIN {X 0,Y 387.69,Z 803.875,A -85,B 0,C 180,E1 -23062.544,E2 -23062.544} C_VEL
LIN {X 0,Y 381.104,Z 828.129,A -85,B 0,C 180,E1 -23063.324,E2 -23063.324} C_VEL
LIN {X 0,Y 374.28,Z 848.813,A -85,B 0,C 180,E1 -23064.172,E2 -23064.172} C_VEL
LIN {X 0,Y 365.745,Z 871.344,A -85,B 0,C 180,E1 -23065.321,E2 -23065.321} C_VEL
LIN {X 0,Y 356.44,Z 892.358,A -85,B 0,C 180,E1 -23066.669,E2 -23066.669} C_VEL
LIN {X 0,Y 346.382,Z 912.781,A -85,B 0,C 180,E1 -23068.256,E2 -23068.256} C_VEL
LIN {X 0,Y 335.391,Z 932.564,A -85,B 0,C 180,E1 -23070.167,E2 -23070.167} C_VEL
LIN {X 0,Y 324.92,Z 949.901,A -85,B 0,C 180,E1 -23072.192,E2 -23072.192} C_VEL
LIN {X 0,Y 312.929,Z 968.085,A -85,B 0,C 180,E1 -23074.797,E2 -23074.797} C_VEL
LIN {X 0,Y 302.254,Z 983.196,A -85,B 0,C 180,E1 -23077.444,E2 -23077.444} C_VEL
LIN {X 0,Y 290.029,Z 999.531,A -85,B 0,C 180,E1 -23080.973,E2 -23080.973} C_VEL
LIN {X 0,Y 279.971,Z 1012.354,A -85,B 0,C 180,E1 -23084.416,E2 -23084.416} C_VEL
LIN {X 0,Y 269.185,Z 1025.802,A -85,B 0,C 180,E1 -23088.893,E2 -23088.893} C_VEL
LIN {X 0,Y 260.773,Z 1036.213,A -85,B 0,C 180,E1 -23093.262,E2 -23093.262} C_VEL
LIN {X 0,Y 252.94,Z 1046.262,A -85,B 0,C 180,E1 -23098.546,E2 -23098.546} C_VEL
LIN {X 0,Y 247.478,Z 1053.723,A -85,B 0,C 180,E1 -23103.613,E2 -23103.613} C_VEL
LIN {X 0,Y 243.363,Z 1060.291,A -85,B 0,C 180,E1 -23109.308,E2 -23109.308} C_VEL
LIN {X 0,Y 241.068,Z 1064.832,A -85,B 0,C 180,E1 -23114.852,E2 -23114.852} C_VEL
LIN {X 0,Y 240.171,Z 1067.628,A -85,B 0,C 180,E1 -23119.687,E2 -23119.687} C_VEL
LIN {X 0,Y 239.975,Z 1069.472,A -85,B 0,C 180,E1 -23124.98,E2 -23124.98} C_VEL
LIN {X 0,Y 240.024,Z 1069.836,A -85,B 0,C 180,E1 -23130,E2 -23130} C_VEL
LIN {X 0,Y 239.982,Z 1069.112,A -85,B 0,C 180,E1 -23134.54,E2 -23134.54} C_VEL
LIN {X 0,Y 240.062,Z 1067.493,A -85,B 0,C 180,E1 -23138.865,E2 -23138.865} C_VEL
LIN {X 0,Y 240.688,Z 1064.623,A -85,B 0,C 180,E1 -23143.697,E2 -23143.697} C_VEL
LIN {X 0,Y 242.774,Z 1059.401,A -85,B 0,C 180,E1 -23149.738,E2 -23149.738} C_VEL
LIN {X 0,Y 245.938,Z 1053.504,A -85,B 0,C 180,E1 -23154.756,E2 -23154.756} C_VEL
LIN {X 0,Y 251.056,Z 1045.569,A -85,B 0,C 180,E1 -23160.121,E2 -23160.121} C_VEL
LIN {X 0,Y 257.954,Z 1035.663,A -85,B 0,C 180,E1 -23165.279,E2 -23165.279} C_VEL
LIN {X 0,Y 266.254,Z 1024.474,A -85,B 0,C 180,E1 -23169.994,E2 -23169.994} C_VEL
LIN {X 0,Y 275.494,Z 1011.927,A -85,B 0,C 180,E1 -23174.175,E2 -23174.175} C_VEL
LIN {X 0,Y 285.04,Z 998.91,A -85,B 0,C 180,E1 -23177.745,E2 -23177.745} C_VEL
LIN {X 0,Y 296.15,Z 983.09,A -85,B 0,C 180,E1 -23181.253,E2 -23181.253} C_VEL
LIN {X 0,Y 306.358,Z 967.847,A -85,B 0,C 180,E1 -23184.021,E2 -23184.021} C_VEL
LIN {X 0,Y 317.965,Z 949.305,A -85,B 0,C 180,E1 -23186.77,E2 -23186.77} C_VEL
LIN {X 0,Y 327.782,Z 932.315,A -85,B 0,C 180,E1 -23188.832,E2 -23188.832} C_VEL
LIN {X 0,Y 338.722,Z 911.666,A -85,B 0,C 180,E1 -23190.9,E2 -23190.9} C_VEL
LIN {X 0,Y 347.872,Z 892.386,A -85,B 0,C 180,E1 -23192.464,E2 -23192.464} C_VEL
LIN {X 0,Y 357.142,Z 870.654,A -85,B 0,C 180,E1 -23193.924,E2 -23193.924} C_VEL
LIN {X 0,Y 364.974,Z 849.253,A -85,B 0,C 180,E1 -23195.069,E2 -23195.069} C_VEL
LIN {X 0,Y 371.657,Z 828.377,A -85,B 0,C 180,E1 -23195.976,E2 -23195.976} C_VEL
LIN {X 0,Y 378.134,Z 803.775,A -85,B 0,C 180,E1 -23196.811,E2 -23196.811} C_VEL
LIN {X 0,Y 382.633,Z 782.361,A -85,B 0,C 180,E1 -23197.372,E2 -23197.372} C_VEL
LIN {X 0,Y 386.671,Z 755.374,A -85,B 0,C 180,E1 -23197.923,E2 -23197.923} C_VEL
LIN {X 0,Y 403.402,Z 568.894,A -85,B 0,C 180,E1 -23200.902,E2 -23200.902} C_VEL
LIN {X 0,Y 398.244,Z 557.633,A -85,B 0,C 180,E1 -23203.668,E2 -23203.668} C_VEL
LIN {X 0,Y 393.971,Z 550.114,A -85,B 0,C 180,E1 -23206.273,E2 -23206.273} C_VEL
LIN {X 0,Y 390.379,Z 543.824,A -85,B 0,C 180,E1 -23208.925,E2 -23208.925} C_VEL
LIN {X 0,Y 387.521,Z 539.169,A -85,B 0,C 180,E1 -23211.543,E2 -23211.543} C_VEL
LIN {X 0,Y 385.179,Z 535.036,A -85,B 0,C 180,E1 -23214.488,E2 -23214.488} C_VEL
LIN {X 0,Y 383.121,Z 530.299,A -85,B 0,C 180,E1 -23221.346,E2 -23221.346} C_VEL
LIN {X 0,Y 385.47,Z 535.482,A -85,B 0,C 180,E1 -23228.352,E2 -23228.352} C_VEL
LIN {X 0,Y 388.46,Z 540.683,A -85,B 0,C 180,E1 -23231.808,E2 -23231.808} C_VEL
LIN {X 0,Y 391.35,Z 545.617,A -85,B 0,C 180,E1 -23234.274,E2 -23234.274} C_VEL
LIN {X 0,Y 395.237,Z 552.118,A -85,B 0,C 180,E1 -23236.952,E2 -23236.952} C_VEL
LIN {X 0,Y 400.428,Z 561.515,A -85,B 0,C 180,E1 -23239.929,E2 -23239.929} C_VEL
LIN {X 0,Y 403.438,Z 567.456,A -85,B 0,C 180,E1 -23241.456,E2 -23241.456} C_VEL
LIN {X 0,Y 387.142,Z 748.135,A -85,B 0,C 180,E1 -23244.331,E2 -23244.331} C_VEL
LIN {X 0,Y 383.184,Z 774.56,A -85,B 0,C 180,E1 -23244.892,E2 -23244.892} C_VEL
LIN {X 0,Y 378.931,Z 795.289,A -85,B 0,C 180,E1 -23245.476,E2 -23245.476} C_VEL
LIN {X 0,Y 372.699,Z 819.594,A -85,B 0,C 180,E1 -23246.354,E2 -23246.354} C_VEL
LIN {X 0,Y 366.226,Z 840.256,A -85,B 0,C 180,E1 -23247.302,E2 -23247.302} C_VEL
LIN {X 0,Y 358.451,Z 861.898,A -85,B 0,C 180,E1 -23248.516,E2 -23248.516} C_VEL
LIN {X 0,Y 349.307,Z 883.51,A -85,B 0,C 180,E1 -23250.014,E2 -23250.014} C_VEL
LIN {X 0,Y 340.037,Z 903.213,A -85,B 0,C 180,E1 -23251.67,E2 -23251.67} C_VEL
LIN {X 0,Y 329.424,Z 923.215,A -85,B 0,C 180,E1 -23253.73,E2 -23253.73} C_VEL
LIN {X 0,Y 319.951,Z 939.603,A -85,B 0,C 180,E1 -23255.761,E2 -23255.761} C_VEL
LIN {X 0,Y 308.213,Z 958.246,A -85,B 0,C 180,E1 -23258.571,E2 -23258.571} C_VEL
LIN {X 0,Y 298.169,Z 973.091,A -85,B 0,C 180,E1 -23261.308,E2 -23261.308} C_VEL
LIN {X 0,Y 286.701,Z 989.113,A -85,B 0,C 180,E1 -23264.93,E2 -23264.93} C_VEL
LIN {X 0,Y 277.303,Z 1001.648,A -85,B 0,C 180,E1 -23268.436,E2 -23268.436} C_VEL
LIN {X 0,Y 267.668,Z 1014.257,A -85,B 0,C 180,E1 -23272.76,E2 -23272.76} C_VEL
LIN {X 0,Y 259.797,Z 1024.412,A -85,B 0,C 180,E1 -23277.134,E2 -23277.134} C_VEL
LIN {X 0,Y 252.758,Z 1033.885,A -85,B 0,C 180,E1 -23282.173,E2 -23282.173} C_VEL
LIN {X 0,Y 247.387,Z 1041.451,A -85,B 0,C 180,E1 -23287.42,E2 -23287.42} C_VEL
LIN {X 0,Y 243.652,Z 1047.556,A -85,B 0,C 180,E1 -23292.814,E2 -23292.814} C_VEL
LIN {X 0,Y 241.317,Z 1052.178,A -85,B 0,C 180,E1 -23298.528,E2 -23298.528} C_VEL
LIN {X 0,Y 240.381,Z 1054.854,A -85,B 0,C 180,E1 -23303.312,E2 -23303.312} C_VEL
LIN {X 0,Y 240.066,Z 1056.49,A -85,B 0,C 180,E1 -23308.091,E2 -23308.091} C_VEL
LIN {X 0,Y 240.014,Z 1057.097,A -85,B 0,C 180,E1 -23313.105,E2 -23313.105} C_VEL
LIN {X 0,Y 240.171,Z 1056.429,A -85,B 0,C 180,E1 -23318.138,E2 -23318.138} C_VEL
LIN {X 0,Y 240.764,Z 1054.748,A -85,B 0,C 180,E1 -23322.959,E2 -23322.959} C_VEL
LIN {X 0,Y 242.354,Z 1051.699,A -85,B 0,C 180,E1 -23328.274,E2 -23328.274} C_VEL
LIN {X 0,Y 245.555,Z 1046.718,A -85,B 0,C 180,E1 -23334.029,E2 -23334.029} C_VEL
LIN {X 0,Y 249.825,Z 1040.987,A -85,B 0,C 180,E1 -23338.966,E2 -23338.966} C_VEL
LIN {X 0,Y 256.801,Z 1032.373,A -85,B 0,C 180,E1 -23344.644,E2 -23344.644} C_VEL
LIN {X 0,Y 264.258,Z 1023.467,A -85,B 0,C 180,E1 -23349.19,E2 -23349.19} C_VEL
LIN {X 0,Y 274.029,Z 1011.899,A -85,B 0,C 180,E1 -23353.89,E2 -23353.89} C_VEL
LIN {X 0,Y 283.806,Z 1000.013,A -85,B 0,C 180,E1 -23357.719,E2 -23357.719} C_VEL
LIN {X 0,Y 295.269,Z 985.638,A -85,B 0,C 180,E1 -23361.467,E2 -23361.467} C_VEL
LIN {X 0,Y 305.967,Z 971.336,A -85,B 0,C 180,E1 -23364.461,E2 -23364.461} C_VEL
LIN {X 0,Y 317.421,Z 955.203,A -85,B 0,C 180,E1 -23367.252,E2 -23367.252} C_VEL
LIN {X 0,Y 328.836,Z 937.519,A -85,B 0,C 180,E1 -23369.719,E2 -23369.719} C_VEL
LIN {X 0,Y 339.38,Z 919.914,A -85,B 0,C 180,E1 -23371.754,E2 -23371.754} C_VEL
LIN {X 0,Y 350.287,Z 899.549,A -85,B 0,C 180,E1 -23373.677,E2 -23373.677} C_VEL
LIN {X 0,Y 358.905,Z 881.731,A -85,B 0,C 180,E1 -23375.07,E2 -23375.07} C_VEL
LIN {X 0,Y 368.941,Z 858.156,A -85,B 0,C 180,E1 -23376.58,E2 -23376.58} C_VEL
LIN {X 0,Y 376.287,Z 838.102,A -85,B 0,C 180,E1 -23377.627,E2 -23377.627} C_VEL
LIN {X 0,Y 383.819,Z 813.925,A -85,B 0,C 180,E1 -23378.642,E2 -23378.642} C_VEL
LIN {X 0,Y 389.378,Z 791.903,A -85,B 0,C 180,E1 -23379.365,E2 -23379.365} C_VEL
LIN {X 0,Y 394.305,Z 767.227,A -85,B 0,C 180,E1 -23379.986,E2 -23379.986} C_VEL
LIN {X 0,Y 397.509,Z 743.917,A -85,B 0,C 180,E1 -23380.423,E2 -23380.423} C_VEL
LIN {X 0,Y 413.233,Z 574.497,A -85,B 0,C 180,E1 -23383.061,E2 -23383.061} C_VEL
LIN {X 0,Y 410.26,Z 568.825,A -85,B 0,C 180,E1 -23384.749,E2 -23384.749} C_VEL
LIN {X 0,Y 408.323,Z 566.877,A -85,B 0,C 180,E1 -23385.847,E2 -23385.847} C_VEL
LIN {X 0,Y 402.936,Z 565.423,A -85,B 0,C 180,E1 -23389.159,E2 -23389.159} C_VEL
LIN {X 0,Y 402.359,Z 564.773,A -85,B 0,C 180,E1 -23389.621,E2 -23389.621} C_VEL
LIN {X 0,Y 399.981,Z 560.605,A -85,B 0,C 180,E1 -23391.953,E2 -23391.953} C_VEL
LIN {X 0,Y 397.86,Z 556.677,A -85,B 0,C 180,E1 -23394.809,E2 -23394.809} C_VEL
LIN {X 0,Y 396.169,Z 552.519,A -85,B 0,C 180,E1 -23400.868,E2 -23400.868} C_VEL
LIN {X 0,Y 398.223,Z 557.306,A -85,B 0,C 180,E1 -23407.43,E2 -23407.43} C_VEL
LIN {X 0,Y 400.781,Z 562.036,A -85,B 0,C 180,E1 -23410.566,E2 -23410.566} C_VEL
LIN {X 0,Y 403.525,Z 566.964,A -85,B 0,C 180,E1 -23413.032,E2 -23413.032} C_VEL
LIN {X 0,Y 406.77,Z 572.828,A -85,B 0,C 180,E1 -23415.395,E2 -23415.395} C_VEL
LIN {X 0,Y 410.341,Z 581.211,A -85,B 0,C 180,E1 -23417.703,E2 -23417.703} C_VEL
LIN {X 0,Y 393.726,Z 755.676,A -85,B 0,C 180,E1 -23420.394,E2 -23420.394} C_VEL
LIN {X 0,Y 389.508,Z 782.287,A -85,B 0,C 180,E1 -23420.909,E2 -23420.909} C_VEL
LIN {X 0,Y 384.811,Z 803.636,A -85,B 0,C 180,E1 -23421.429,E2 -23421.429} C_VEL
LIN {X 0,Y 377.998,Z 828.265,A -85,B 0,C 180,E1 -23422.206,E2 -23422.206} C_VEL
LIN {X 0,Y 371.058,Z 848.906,A -85,B 0,C 180,E1 -23423.039,E2 -23423.039} C_VEL
LIN {X 0,Y 362.252,Z 871.633,A -85,B 0,C 180,E1 -23424.182,E2 -23424.182} C_VEL
LIN {X 0,Y 352.801,Z 892.535,A -85,B 0,C 180,E1 -23425.507,E2 -23425.507} C_VEL
LIN {X 0,Y 342.316,Z 913.337,A -85,B 0,C 180,E1 -23427.108,E2 -23427.108} C_VEL
LIN {X 0,Y 331.006,Z 933.122,A -85,B 0,C 180,E1 -23429.013,E2 -23429.013} C_VEL
LIN {X 0,Y 319.94,Z 950.948,A -85,B 0,C 180,E1 -23431.095,E2 -23431.095} C_VEL
LIN {X 0,Y 307.654,Z 968.923,A -85,B 0,C 180,E1 -23433.694,E2 -23433.694} C_VEL
LIN {X 0,Y 296.416,Z 984.325,A -85,B 0,C 180,E1 -23436.42,E2 -23436.42} C_VEL
LIN {X 0,Y 284.108,Z 1000.112,A -85,B 0,C 180,E1 -23439.894,E2 -23439.894} C_VEL
LIN {X 0,Y 274.242,Z 1012.221,A -85,B 0,C 180,E1 -23443.18,E2 -23443.18} C_VEL
LIN {X 0,Y 262.999,Z 1025.652,A -85,B 0,C 180,E1 -23447.706,E2 -23447.706} C_VEL
LIN {X 0,Y 254.566,Z 1035.589,A -85,B 0,C 180,E1 -23451.927,E2 -23451.927} C_VEL
LIN {X 0,Y 246.508,Z 1045.405,A -85,B 0,C 180,E1 -23457.102,E2 -23457.102} C_VEL
LIN {X 0,Y 240.341,Z 1053.235,A -85,B 0,C 180,E1 -23462.497,E2 -23462.497} C_VEL
LIN {X 0,Y 235.845,Z 1059.872,A -85,B 0,C 180,E1 -23468.355,E2 -23468.355} C_VEL
LIN {X 0,Y 233.202,Z 1064.635,A -85,B 0,C 180,E1 -23474.328,E2 -23474.328} C_VEL
LIN {X 0,Y 232.206,Z 1067.427,A -85,B 0,C 180,E1 -23479.33,E2 -23479.33} C_VEL
LIN {X 0,Y 231.976,Z 1069.266,A -85,B 0,C 180,E1 -23484.807,E2 -23484.807} C_VEL
LIN {X 0,Y 232.019,Z 1069.641,A -85,B 0,C 180,E1 -23489.753,E2 -23489.753} C_VEL
LIN {X 0,Y 231.984,Z 1068.958,A -85,B 0,C 180,E1 -23494.45,E2 -23494.45} C_VEL
LIN {X 0,Y 232.065,Z 1067.379,A -85,B 0,C 180,E1 -23498.923,E2 -23498.923} C_VEL
LIN {X 0,Y 232.701,Z 1064.624,A -85,B 0,C 180,E1 -23503.808,E2 -23503.808} C_VEL
LIN {X 0,Y 234.7,Z 1059.909,A -85,B 0,C 180,E1 -23509.69,E2 -23509.69} C_VEL
LIN {X 0,Y 238.268,Z 1053.553,A -85,B 0,C 180,E1 -23515.343,E2 -23515.343} C_VEL
LIN {X 0,Y 243.373,Z 1046.025,A -85,B 0,C 180,E1 -23520.627,E2 -23520.627} C_VEL
LIN {X 0,Y 250.514,Z 1036.315,A -85,B 0,C 180,E1 -23525.925,E2 -23525.925} C_VEL
LIN {X 0,Y 258.183,Z 1026.358,A -85,B 0,C 180,E1 -23530.297,E2 -23530.297} C_VEL
LIN {X 0,Y 268.617,Z 1012.911,A -85,B 0,C 180,E1 -23535.011,E2 -23535.011} C_VEL
LIN {X 0,Y 277.893,Z 1000.729,A -85,B 0,C 180,E1 -23538.453,E2 -23538.453} C_VEL
LIN {X 0,Y 289.353,Z 985.184,A -85,B 0,C 180,E1 -23542.041,E2 -23542.041} C_VEL
LIN {X 0,Y 299.7,Z 970.261,A -85,B 0,C 180,E1 -23544.825,E2 -23544.825} C_VEL
LIN {X 0,Y 311.165,Z 952.835,A -85,B 0,C 180,E1 -23547.513,E2 -23547.513} C_VEL
LIN {X 0,Y 322.546,Z 933.775,A -85,B 0,C 180,E1 -23549.871,E2 -23549.871} C_VEL
LIN {X 0,Y 333.349,Z 914.165,A -85,B 0,C 180,E1 -23551.868,E2 -23551.868} C_VEL
LIN {X 0,Y 343.386,Z 893.65,A -85,B 0,C 180,E1 -23553.544,E2 -23553.544} C_VEL
LIN {X 0,Y 352.222,Z 873.559,A -85,B 0,C 180,E1 -23554.901,E2 -23554.901} C_VEL
LIN {X 0,Y 360.979,Z 850.598,A -85,B 0,C 180,E1 -23556.146,E2 -23556.146} C_VEL
LIN {X 0,Y 367.442,Z 830.991,A -85,B 0,C 180,E1 -23557.001,E2 -23557.001} C_VEL
LIN {X 0,Y 374.212,Z 806.578,A -85,B 0,C 180,E1 -23557.847,E2 -23557.847} C_VEL
LIN {X 0,Y 379.062,Z 784.332,A -85,B 0,C 180,E1 -23558.433,E2 -23558.433} C_VEL
LIN {X 0,Y 383.117,Z 759.514,A -85,B 0,C 180,E1 -23558.951,E2 -23558.951} C_VEL
